// TwinCAT 3 PLC project Library
// Title: lcls-twincat-motion-abstraction
// Company: SLAC
// Author: YS Mandza
// ProjectVersion: 1.0.0
// Description: Motion Abstraction
// ProgramVersion: 3.1.4026.17
// libraries:
//   LCLS General, * (SLAC)
//   Tc2_EtherCAT, * (Beckhoff Automation GmbH)
//   Tc2_MC2, * (Beckhoff Automation GmbH)
//   Tc2_Standard, * (Beckhoff Automation GmbH)
//   Tc2_System, * (Beckhoff Automation GmbH)
//   Tc2_Utilities, * (Beckhoff Automation GmbH)
//   TcUnit, * (www.tcunit.org)
// project tree:
//   / DemoTask.TcTTO, PlcTask.TcTTO, UnitTestTask.TcTTO (not stored)
//   DUTs/ E_LCLSMotionError.TcDUT (not stored), E_MotionLogLevel.TcDUT, MOTION_LOGGER_MSG.TcDUT, ST_ExtendedMotionStatus.TcDUT, E_HomeStates.TcDUT (not stored), E_Module.TcDUT (not stored), ST_MotionStatus.TcDUT (not stored), ENUM_StageEnableMode.TcDUT (not stored), E_DS402HomingMethod.TcDUT (not stored), E_DS402OpMode.TcDUT (not stored), E_EpicsHomeCmd.TcDUT, E_EpicsMotorCmd.TcDUT, E_MoveMode.TcDUT (not stored), E_MoveState.TcDUT, E_StageBrakeMode.TcDUT, E_StageEnableMode.TcDUT (not stored), ST_AxisParameterSetExposed.TcDUT (not stored), ST_DS402Drive.TcDUT, ST_DS402DriveStatus.TcDUT (not stored), ST_AxisStatus.TcDUT (not stored), ST_MotionCommand.TcDUT (not stored), ST_MotionLogMessage.TcDUT, ST_MoveRequestStatus.TcDUT (not stored)
//   POUs/FBs/Common/ FB_EncoderScaling.TcPOU (not stored), FB_EpicsMotionParamsStatus.TcPOU (not stored), FB_EpicsMoveRequest.TcPOU, FB_LimSwStatus.TcPOU (not stored), FB_MotionDrive.TcPOU, FB_MotionDriveStateMachine.TcPOU (not stored), FB_MotionInterlocksCommon.TcPOU (not stored), FB_MotionInterlocksLimSw.TcPOU (not stored), FB_MotionLogger.TcPOU, FB_PersistentDataStorage.TcPOU (not stored)
//   POUs/FBs/Containers/ FB_MotionStageNC.TcPOU
//   POUs/FBs/DS402/ FB_HomeDS402.TcPOU (not stored) (excluded from build)
//   POUs/FBs/NC/ FB_AxisStatusNC.TcPOU (not stored) (excluded from build), FB_BacklashCompensationNC.TcPOU (not stored), FB_BrakeNC.TcPOU (not stored), FB_HaltNC.TcPOU (not stored), FB_HomeNC.TcPOU (not stored), FB_MotionAxisNC.TcPOU (not stored), FB_MoveAbsoluteNC.TcPOU (not stored), FB_ParamsSaveRestoreNC.TcPOU, FB_PowerInterlockNC.TcPOU (not stored), FB_PowerNC.TcPOU (not stored), FB_ReadParameterNC.TcPOU (not stored), FB_ResetNC.TcPOU (not stored), FB_WriteParameterNC.TcPOU (not stored)
//   POUs/ITFs/ I_AxisStatus.TcIO (not stored), I_BacklashCompensation.TcIO (not stored), I_Brake.TcIO (not stored), I_DS402GenericDrive.TcIO (not stored), I_EncoderScaling.TcIO (not stored), I_EpicsMotionParamsStatus.TcIO (not stored), I_Error.TcIO (not stored), I_Halt.TcIO, I_Home.TcIO (not stored), I_HomeDS402.TcIO (not stored), I_LimSwStatus.TcIO (not stored), I_MotionAxis.TcIO (not stored), I_MotionAxisDS402.TcIO (not stored), I_MotionDrive.TcIO (not stored), I_MotionInterlocks.TcIO (not stored), I_MotionInterlocksCommon.TcIO (not stored), I_MotionLogger.TcIO, I_MotionStage.TcIO (not stored), I_MoveAbsolute.TcIO (not stored), I_MoveRequest.TcIO, I_ParamsSaveRestore.TcIO, I_PersistentDataStorage.TcIO (not stored), I_Power.TcIO (not stored), I_ReadParameter.TcIO (not stored), I_Reset.TcIO (not stored), I_StateMachine.TcIO (not stored), I_Status.TcIO (not stored), I_StatusEx.TcIO (not stored), I_WriteParameter.TcIO (not stored)
//   Test/Containers/ FB_MotionStageNC_Test.TcPOU
//   Test/Interlok/ FB_MotionInterlocksCommon_Test.TcPOU, FB_MotionInterlocksLimSw_Test.TcPOU
//   Test/ HARD_TEST.TcPOU (not stored), PRG_TEST.TcPOU (not stored), CONTAINER_TEST.TcPOU (not stored)
//   Test/Orchetration/ FB_BrakeNC_Test.TcPOU (not stored), FB_MotionDriveStateMachine_Test.TcPOU, FB_MotionDrive_Test.TcPOU (not stored), FB_MoveRequest_Test.TcPOU
//   Test/NC/ FB_NcMotionBlocks_Test.TcPOU, FB_MotionAxisNC_Test.TcPOU
//   Test/TestDouble/ FB_AxisStatusNC_TestDouble.TcPOU (not stored), FB_BacklashCompensationNC_TestDouble.TcPOU (not stored), FB_Brake_TestDouble.TcPOU (not stored), FB_EncoderScalingNC_TestDouble.TcPOU (not stored), FB_EpicsMotionParamsStatus_TestDouble.TcPOU (not stored), FB_HaltNC_TestDouble.TcPOU, FB_HomeNC_TestDouble.TcPOU (not stored), FB_LimSwStatus_testDouble.TcPOU (not stored), FB_MotionAxisDS402_TestDouble.TcPOU, FB_MotionAxisNC_TestDouble.TcPOU (not stored), FB_StateMachine_TestDouble.TcPOU (not stored), FB_MotionInterlocksCommon_TestDouble.TcPOU (not stored), FB_MotionInterlocksLimSw_TestDouble.TcPOU, FB_MotionLogger_TestDouble.TcPOU, FB_MoveAbsoluteNC_TestDouble.TcPOU, FB_MoveRequest_TestDouble.TcPOU (not stored), FB_ParamSaveRestoreNC_TestDouble.TcPOU, FB_PersistentDataStorage_TestDouble.TcPOU, FB_PowerNC_TestDouble.TcPOU (not stored), FB_ReadParameterNC_TestDouble.TcPOU (not stored), FB_ResetNC_TestDouble.TcPOU, FB_WriteParameterNC_TestDouble.TcPOU (not stored)
//   Test/Utils/ FB_MotionLogger_Test.TcPOU (not stored)
//   VISUs/ motion.TcCD (not stored)
// real-time tasks:
//   TASK PlcTask: cycle T#10ms, priority 1, ADS port 350
//   TASK UnitTestTask: cycle T#10ms, priority 20, ADS port 351
//   TASK Demo: cycle T#10ms, priority 2, ADS port 352
// motion (NC):
//   TASK NC-Task 1 SAF: cycle T#2ms, priority 4, ADS port 501
//   TASK NC-Task 1 SVB: cycle T#10ms, priority 8, ADS port 511
//   AXIS Axis_HomeNC_Test8 (id 15)
//     OtherSettings: AllowMotionCmdToSlave=true
//     encoder EncType=1
//     drive DrvType=5
//       Analog: TorqueSetpointScale=10, ScaleFactorActTorque=0.1
//       TimeComp: TaskDelayCycles=1
//     controller CtrType=1
//       CtrPara: PriorControlFactor=1
//         Observer: BandWidth=20
//   AXIS Axis_HomeNC_Test7 (id 14)
//     OtherSettings: AllowMotionCmdToSlave=true
//     encoder EncType=1
//     drive DrvType=5
//       Analog: TorqueSetpointScale=10, ScaleFactorActTorque=0.1
//       TimeComp: TaskDelayCycles=1
//     controller CtrType=1
//       CtrPara: PriorControlFactor=1
//         Observer: BandWidth=20
//   AXIS Axis_HomeNC_Test6 (id 2)
//     OtherSettings: AllowMotionCmdToSlave=true
//     encoder EncType=1
//     drive DrvType=5
//       Analog: TorqueSetpointScale=10, ScaleFactorActTorque=0.1
//       TimeComp: TaskDelayCycles=1
//     controller CtrType=1
//       CtrPara: PriorControlFactor=1
//         Observer: BandWidth=20
//   AXIS Axis_HomeNC_Test5 (id 7)
//     OtherSettings: AllowMotionCmdToSlave=true
//     encoder EncType=1
//     drive DrvType=5
//       Analog: TorqueSetpointScale=10, ScaleFactorActTorque=0.1
//       TimeComp: TaskDelayCycles=1
//     controller CtrType=1
//       CtrPara: PriorControlFactor=1
//         Observer: BandWidth=20
//   AXIS Axis_HomeNC_Test4 (id 6)
//     OtherSettings: AllowMotionCmdToSlave=true
//     encoder EncType=1
//     drive DrvType=5
//       Analog: TorqueSetpointScale=10, ScaleFactorActTorque=0.1
//       TimeComp: TaskDelayCycles=1
//     controller CtrType=1
//       CtrPara: PriorControlFactor=1
//         Observer: BandWidth=20
//   AXIS Axis_HomeNC_Test3 (id 5)
//     OtherSettings: AllowMotionCmdToSlave=true
//     encoder EncType=1
//     drive DrvType=5
//       Analog: TorqueSetpointScale=10, ScaleFactorActTorque=0.1
//       TimeComp: TaskDelayCycles=1
//     controller CtrType=1
//       CtrPara: PriorControlFactor=1
//         Observer: BandWidth=20
//   AXIS Axis_HomeNC_Test2 (id 4)
//     Velo: RefSearch=500, RefSync=500
//     OtherSettings: AllowMotionCmdToSlave=true
//     encoder EncType=1
//     drive DrvType=5
//       Analog: TorqueSetpointScale=10, ScaleFactorActTorque=0.1
//       TimeComp: TaskDelayCycles=1
//     controller CtrType=1
//       CtrPara: PriorControlFactor=1
//         Observer: BandWidth=20
//   AXIS Axis_HomeNC_Test1 (id 3)
//     OtherSettings: AllowMotionCmdToSlave=true
//     encoder EncType=1
//     drive DrvType=5
//       Analog: TorqueSetpointScale=10, ScaleFactorActTorque=0.1
//       TimeComp: TaskDelayCycles=1
//     controller CtrType=1
//       CtrPara: PriorControlFactor=1
//         Observer: BandWidth=20
//   AXIS Axis_McMotionBlocks_Test1 (id 9)
//     OtherSettings: AllowMotionCmdToSlave=true
//     encoder EncType=1
//     drive DrvType=5
//       Analog: TorqueSetpointScale=10, ScaleFactorActTorque=0.1
//       TimeComp: TaskDelayCycles=1
//     controller CtrType=1
//       CtrPara: PriorControlFactor=1
//         Observer: BandWidth=20
//   AXIS Axis_McMotionBlocks_Test2 (id 10)
//     OtherSettings: AllowMotionCmdToSlave=true
//     encoder EncType=1
//     drive DrvType=5
//       Analog: TorqueSetpointScale=10, ScaleFactorActTorque=0.1
//       TimeComp: TaskDelayCycles=1
//     controller CtrType=1
//       CtrPara: PriorControlFactor=1
//         Observer: BandWidth=20
//   AXIS Axis_McMotionBlocks_Test3 (id 11)
//     OtherSettings: AllowMotionCmdToSlave=true
//     encoder EncType=1
//     drive DrvType=5
//       Analog: TorqueSetpointScale=10, ScaleFactorActTorque=0.1
//       TimeComp: TaskDelayCycles=1
//     controller CtrType=1
//       CtrPara: PriorControlFactor=1
//         Observer: BandWidth=20
//   AXIS Axis_McMotionBlocks_Test4 (id 12)
//     OtherSettings: AllowMotionCmdToSlave=true
//     encoder EncType=1
//     drive DrvType=5
//       Analog: TorqueSetpointScale=10, ScaleFactorActTorque=0.1
//       TimeComp: TaskDelayCycles=1
//     controller CtrType=1
//       CtrPara: PriorControlFactor=1
//         Observer: BandWidth=20
//   AXIS Axis_McMotionBlocks_Test8 (id 17)
//     OtherSettings: AllowMotionCmdToSlave=true
//     encoder EncType=1
//       ActPosCorrection: Enable=true
//     drive DrvType=5
//       Analog: TorqueSetpointScale=10, ScaleFactorActTorque=0.1
//       TimeComp: TaskDelayCycles=1
//     controller CtrType=1
//       CtrPara: PriorControlFactor=1
//         Observer: BandWidth=20
//   AXIS Axis_McMotionBlocks_Test7 (id 1)
//     OtherSettings: AllowMotionCmdToSlave=true
//     encoder EncType=1
//       ActPosCorrection: Enable=true
//     drive DrvType=5
//       Analog: TorqueSetpointScale=10, ScaleFactorActTorque=0.1
//       TimeComp: TaskDelayCycles=1
//     controller CtrType=1
//       CtrPara: PriorControlFactor=1
//         Observer: BandWidth=20
//   AXIS Axis_McMotionBlocks_Test6 (id 16)
//     OtherSettings: AllowMotionCmdToSlave=true
//     encoder EncType=1
//       ActPosCorrection: Enable=true
//     drive DrvType=5
//       Analog: TorqueSetpointScale=10, ScaleFactorActTorque=0.1
//       TimeComp: TaskDelayCycles=1
//     controller CtrType=1
//       CtrPara: PriorControlFactor=1
//         Observer: BandWidth=20
//   AXIS Axis_McMotionBlocks_Test5 (id 13)
//     OtherSettings: AllowMotionCmdToSlave=true
//     encoder EncType=1
//     drive DrvType=5
//       Analog: TorqueSetpointScale=10, ScaleFactorActTorque=0.1
//       TimeComp: TaskDelayCycles=1
//     controller CtrType=1
//       CtrPara: PriorControlFactor=1
//         Observer: BandWidth=20
//   AXIS Axis_Hard_Test (id 8)
//     Velo: RefSync=100
//     OtherSettings: AllowMotionCmdToSlave=true
//     encoder EncType=1
//       ActPosCorrection: Enable=true
//     drive DrvType=5
//       Analog: TorqueSetpointScale=10, ScaleFactorActTorque=0.1
//       TimeComp: TaskDelayCycles=1
//     controller CtrType=1
//       CtrPara: PriorControlFactor=1
//         Observer: BandWidth=20
// variable links:
//   motion/motion Instance <-> NC-Task 1 SAF/Axes/Axis_Hard_Test
//     DemoTask Inputs/NcAxis_GVL.NC.NcToPlc <-> Outputs/ToPlc
//     DemoTask Outputs/NcAxis_GVL.NC.PlcToNc <-> Inputs/FromPlc
//   motion/motion Instance <-> NC-Task 1 SAF/Axes/Axis_HomeNC_Test1
//     UnitTestTask Inputs/PRG_TEST.fb_HomeNC_Test.fbAxisRef[1].NcToPlc <-> Outputs/ToPlc
//     UnitTestTask Outputs/PRG_TEST.fb_HomeNC_Test.fbAxisRef[1].PlcToNc <-> Inputs/FromPlc
//   motion/motion Instance <-> NC-Task 1 SAF/Axes/Axis_HomeNC_Test2
//     UnitTestTask Inputs/PRG_TEST.fb_HomeNC_Test.fbAxisRef[2].NcToPlc <-> Outputs/ToPlc
//     UnitTestTask Outputs/PRG_TEST.fb_HomeNC_Test.fbAxisRef[2].PlcToNc <-> Inputs/FromPlc
//   motion/motion Instance <-> NC-Task 1 SAF/Axes/Axis_HomeNC_Test3
//     UnitTestTask Inputs/PRG_TEST.fb_HomeNC_Test.fbAxisRef[3].NcToPlc <-> Outputs/ToPlc
//     UnitTestTask Outputs/PRG_TEST.fb_HomeNC_Test.fbAxisRef[3].PlcToNc <-> Inputs/FromPlc
//   motion/motion Instance <-> NC-Task 1 SAF/Axes/Axis_HomeNC_Test4
//     UnitTestTask Inputs/PRG_TEST.fb_HomeNC_Test.fbAxisRef[4].NcToPlc <-> Outputs/ToPlc
//     UnitTestTask Outputs/PRG_TEST.fb_HomeNC_Test.fbAxisRef[4].PlcToNc <-> Inputs/FromPlc
//   motion/motion Instance <-> NC-Task 1 SAF/Axes/Axis_HomeNC_Test5
//     UnitTestTask Inputs/PRG_TEST.fb_HomeNC_Test.fbAxisRef[5].NcToPlc <-> Outputs/ToPlc
//     UnitTestTask Outputs/PRG_TEST.fb_HomeNC_Test.fbAxisRef[5].PlcToNc <-> Inputs/FromPlc
//   motion/motion Instance <-> NC-Task 1 SAF/Axes/Axis_HomeNC_Test6
//     UnitTestTask Inputs/PRG_TEST.fb_HomeNC_Test.fbAxisRef[6].NcToPlc <-> Outputs/ToPlc
//     UnitTestTask Outputs/PRG_TEST.fb_HomeNC_Test.fbAxisRef[6].PlcToNc <-> Inputs/FromPlc
//   motion/motion Instance <-> NC-Task 1 SAF/Axes/Axis_HomeNC_Test7
//     UnitTestTask Inputs/PRG_TEST.fb_HomeNC_Test.fbAxisRef[7].NcToPlc <-> Outputs/ToPlc
//     UnitTestTask Outputs/PRG_TEST.fb_HomeNC_Test.fbAxisRef[7].PlcToNc <-> Inputs/FromPlc
//   motion/motion Instance <-> NC-Task 1 SAF/Axes/Axis_HomeNC_Test8
//     UnitTestTask Inputs/PRG_TEST.fb_HomeNC_Test.fbAxisRef[8].NcToPlc <-> Outputs/ToPlc
//     UnitTestTask Outputs/PRG_TEST.fb_HomeNC_Test.fbAxisRef[8].PlcToNc <-> Inputs/FromPlc
//   motion/motion Instance <-> NC-Task 1 SAF/Axes/Axis_McMotionBlocks_Test1
//     UnitTestTask Inputs/PRG_TEST.fb_McMotionBlocks_Test.fbAxisRef[1].NcToPlc <-> Outputs/ToPlc
//     UnitTestTask Outputs/PRG_TEST.fb_McMotionBlocks_Test.fbAxisRef[1].PlcToNc <-> Inputs/FromPlc
//   motion/motion Instance <-> NC-Task 1 SAF/Axes/Axis_McMotionBlocks_Test2
//     UnitTestTask Inputs/PRG_TEST.fb_McMotionBlocks_Test.fbAxisRef[2].NcToPlc <-> Outputs/ToPlc
//     UnitTestTask Outputs/PRG_TEST.fb_McMotionBlocks_Test.fbAxisRef[2].PlcToNc <-> Inputs/FromPlc
//   motion/motion Instance <-> NC-Task 1 SAF/Axes/Axis_McMotionBlocks_Test3
//     UnitTestTask Inputs/PRG_TEST.fb_McMotionBlocks_Test.fbAxisRef[3].NcToPlc <-> Outputs/ToPlc
//     UnitTestTask Outputs/PRG_TEST.fb_McMotionBlocks_Test.fbAxisRef[3].PlcToNc <-> Inputs/FromPlc
//   motion/motion Instance <-> NC-Task 1 SAF/Axes/Axis_McMotionBlocks_Test4
//     UnitTestTask Inputs/PRG_TEST.fb_McMotionBlocks_Test.fbAxisRef[4].NcToPlc <-> Outputs/ToPlc
//     UnitTestTask Outputs/PRG_TEST.fb_McMotionBlocks_Test.fbAxisRef[4].PlcToNc <-> Inputs/FromPlc
//   motion/motion Instance <-> NC-Task 1 SAF/Axes/Axis_McMotionBlocks_Test5
//     UnitTestTask Inputs/PRG_TEST.fb_McMotionBlocks_Test.fbAxisRef[5].NcToPlc <-> Outputs/ToPlc
//     UnitTestTask Outputs/PRG_TEST.fb_McMotionBlocks_Test.fbAxisRef[5].PlcToNc <-> Inputs/FromPlc
//   motion/motion Instance <-> NC-Task 1 SAF/Axes/Axis_McMotionBlocks_Test6
//     UnitTestTask Inputs/PRG_TEST.fb_McMotionBlocks_Test.fbAxisRef[6].NcToPlc <-> Outputs/ToPlc
//     UnitTestTask Outputs/PRG_TEST.fb_McMotionBlocks_Test.fbAxisRef[6].PlcToNc <-> Inputs/FromPlc
//   motion/motion Instance <-> NC-Task 1 SAF/Axes/Axis_McMotionBlocks_Test7
//     UnitTestTask Inputs/PRG_TEST.fb_McMotionBlocks_Test.fbAxisRef[7].NcToPlc <-> Outputs/ToPlc
//     UnitTestTask Outputs/PRG_TEST.fb_McMotionBlocks_Test.fbAxisRef[7].PlcToNc <-> Inputs/FromPlc
//   motion/motion Instance <-> NC-Task 1 SAF/Axes/Axis_McMotionBlocks_Test8
//     UnitTestTask Inputs/PRG_TEST.fb_McMotionBlocks_Test.fbAxisRef[8].NcToPlc <-> Outputs/ToPlc
//     UnitTestTask Outputs/PRG_TEST.fb_McMotionBlocks_Test.fbAxisRef[8].PlcToNc <-> Inputs/FromPlc

CONFIGURATION Library
    RESOURCE PLC ON TwinCAT3
        TASK DemoTask(INTERVAL := T#10ms, PRIORITY := 2);
        TASK PlcTask(INTERVAL := T#10ms, PRIORITY := 1);
        PROGRAM CONTAINER_TEST WITH DemoTask : CONTAINER_TEST;
        PROGRAM HARD_TEST WITH PlcTask : HARD_TEST;
    END_RESOURCE
END_CONFIGURATION

// ---- DUTs/E_MotionLogLevel.TcDUT
{attribute 'qualified_only'}
{attribute 'strict'}
{attribute 'to_string'}
TYPE E_MotionLogLevel :
(
	WARNING := 0,
	ERROR := 1,
	INFO := 2
);
END_TYPE

// ---- DUTs/MOTION_LOGGER_MSG.TcDUT
TYPE MOTION_LOGGER_MSG : STRING(128); END_TYPE

// ---- DUTs/ST_ExtendedMotionStatus.TcDUT
TYPE ST_ExtendedMotionStatus :
STRUCT
	bMotionAxisError : BOOL;
	nMotionAxisErrorId : UDINT;
	bInterlocksError : BOOL;
	nInterlocksError : UDINT;
	eDriveState : E_MoveState;
	bDriveWatchDogStatus : BOOL;
	bAbortDone : BOOL;
	bAborted : BOOL;
	bLimHomeDone : BOOL;
	bNewMoveReq : BOOL;
	bExecute : BOOL;
	bEnable : BOOL;
	bIdling : BOOL;
END_STRUCT
END_TYPE

// ---- DUTs/E_EpicsHomeCmd.TcDUT
{attribute 'qualified_only'}
{attribute 'strict'}
TYPE E_EpicsHomeCmd :
    // Defines the valid options for homing in FB_MotionStage
(
    LOW_LIMIT := 1, // Low limit switch
    HIGH_LIMIT := 2, // High limit switch
    HOME_VIA_LOW := 3, // Home switch via low switch
    HOME_VIA_HIGH := 4, // Home switch via high switch
    ABSOLUTE_SET := 15, // Set here to be fHomePosition
    // MCS2
    AUTOZERO := -1,
    CURRENT_POSITION_METHOD := 37,
    NONE := -99 // Do not home, ever
) INT := NONE;
END_TYPE

// ---- DUTs/E_EpicsMotorCmd.TcDUT
{attribute 'qualified_only'}
{attribute 'strict'}
TYPE E_EpicsMotorCmd :
    // Defines valid EPICS commands for nCommand
(
    JOG := 0,
    MOVE_VELOCITY := 1,
    MOVE_RELATIVE := 2,
    MOVE_ABSOLUTE := 3,
    MOVE_MODULO := 4,
    HOME := 10,
    GEAR := 30
)INT;
END_TYPE

// ---- DUTs/E_MoveState.TcDUT
{attribute 'qualified_only'}
{attribute 'to_string'}
TYPE E_MoveState :
(
    IDLING:=0,
    INIT:=10,
    STARTED:=20,
    IN_PROGRESS :=30,
    REACHED:=40,
    INTERRUPTED:=50,
    DONE:=60,
    ERROR:=-99
) INT;
END_TYPE

// ---- DUTs/E_StageBrakeMode.TcDUT
{attribute 'qualified_only'}
{attribute 'strict'}
TYPE E_StageBrakeMode :
    // Defines when to send the brake disengage signal in FB_MotionStage
(
    IF_ENABLED := 0, // Disengage brake when the motor is enabled
    IF_MOVING, // Disengage brake when the motor is moving
    NO_BRAKE // Do not change the brake state in FB_MotionStage
)INT;
END_TYPE

// ---- DUTs/ST_DS402Drive.TcDUT
TYPE ST_DS402Drive:
STRUCT
    (* Global variables for the TPDO data from the drive. Each one is linked to the respective TPDO channel. *)
    stDriveStatus 			AT %I*	: 	ST_DS402DriveStatus;
    nModeOfOperationDisplay AT %I*	: 	SINT;
    //nActualPosition 		AT %I*	: 	DINT;
    (*CSP drive mode*)
    nFollowingError 		AT %I*	: 	DINT;
    (* Global variables for the RPDO data to the drive. Each one is linked to the respective RPDO channel. *)
    //nDS402DriveControl		AT %Q*	:	UINT;
    // Connected to NC task Ctrl 1 and Ctrl 2
       nDS402DriveControlNC	AT %I*	:	UINT;
    // connected to I/O Task 'Control Word'
       nDS402DriveControl		AT %Q*	:	UINT;
    //nTargetPositionTmp 		AT %I* 	: 	DINT;
    nTargetPosition 		AT %Q* 	: 	DINT;
    nModeOfOperationNC 	AT %I* 	: 	SINT;
    nModeOfOperation 		AT %Q* 	: 	SINT;
    (* Global variables for the RPDO data to the drive. Each one is linked to the respective RPDO channel. *)
    nProfilVelocity 		AT %Q* 	: 	DINT;
    nProfilAcceleration		AT %Q* 	: 	DINT;
    nProfilDecceleration	AT %Q* 	: 	DINT;
    nVelocityActualValue	AT %Q* 	: 	DINT;
    (* Global variables for the TPDO data from the drive. Each one is linked to the respective TPDO channel. *)
    nScantargetPosition		AT %Q*	: 	DINT;
    uScantargetVelocity		AT %Q*	: 	ULINT;

    {attribute 'pytmc' := '
        pv: PLC:nChanStep
        io: io
        field: DESC SmartAct: Open Loop Step Count
    '}
    nChanStep			: DINT;

    {attribute 'pytmc' := '
        pv: PLC:nChanStepFreq
        io: io
        field: DESC SmartAct: Open Loop Step Freq
    '}
    nChanStepFreq		: UINT;

    {attribute 'pytmc' := '
        pv: PLC:nChanStepAmp
        io: io
        field: DESC SmartAct: Open Loop Step Amp
    '}
    nChanStepAmp		: UINT;

    // timeout for holding actual position in close loop mode
    {attribute 'pytmc' := '
        pv: PLC:nHoldTime
        io: io
        field: DESC SmartAct: Set servo mode hold time
    '}
    nHoldTime						: UDINT := 10000;

    {attribute 'pytmc' := '
        pv: PLC:bServo
        io: io
        field: ZNAM DISABLE
        field: ONAM ENABLE
        field: DESC Used to disable close loop mode
    '}
    bServo							: BOOL := TRUE;

    (* NetId of EtherCAT Master *)
    arNetId  				AT %I*	: 	AMSNETID;
    (* Port Number of EtherCAT Slave *)
    nSlaveAddr 				AT %I* 	: 	UINT;

END_STRUCT
END_TYPE

// ---- DUTs/ST_MotionLogMessage.TcDUT
TYPE ST_MotionLogMessage :
STRUCT
    sSource : STRING(64);
    sMessage : MOTION_LOGGER_MSG;
    sTimestamp : STRING(16);
    eLevel : E_MotionLogLevel;
END_STRUCT
END_TYPE

// ---- POUs/ITFs/I_Halt.TcIO
INTERFACE I_Halt EXTENDS I_StatusEx

METHOD ClearStatus
VAR_INPUT
END_VAR
END_METHOD

PROPERTY CommandHalt : BOOL
SET
END_SET
END_PROPERTY

METHOD Halt
VAR_INPUT
    Deceleration : LREAL := 0.0;
    Jerk : LREAL := 0.0;
    BufferMode	: MC_BufferMode := MC_BufferMode.MC_Aborting;
END_VAR
END_METHOD

END_INTERFACE

// ---- POUs/ITFs/I_MotionLogger.TcIO
INTERFACE I_MotionLogger

METHOD Clear
VAR_INPUT
END_VAR
END_METHOD

METHOD ErrorCodeLookup : STRING
VAR_INPUT
	 nErrorId: UDINT;
END_VAR
END_METHOD

METHOD GetAllMessages : STRING(1024)
END_METHOD

METHOD GetMessageCount : UINT
VAR_OUTPUT
    nCount : UINT;
END_VAR
END_METHOD

METHOD Logger
VAR_INPUT
    Message : STRING;
    Level   : E_MotionLogLevel := E_MotionLogLevel.INFO;
    Source  : STRING := '';
END_VAR
END_METHOD

PROPERTY Name : STRING
GET
END_GET
END_PROPERTY

END_INTERFACE

// ---- POUs/ITFs/I_MoveRequest.TcIO
INTERFACE I_MoveRequest

METHOD ClearMoveRequest
END_METHOD

METHOD ClearMoveRequestErrors
VAR_INPUT
END_VAR
END_METHOD

PROPERTY EnableMode : ENUM_StageEnableMode
GET
END_GET
SET
END_SET
END_PROPERTY

METHOD InitMoveRequest
VAR_INPUT
END_VAR
END_METHOD

METHOD IsValidHomeCmd : BOOL
VAR_INPUT
    CmdData : INT;
END_VAR
END_METHOD

METHOD MoveRequest
VAR_INPUT
	// From Axis through the drive
	EnableDone	: BOOL;
	// From Interlock through the drive
	MoveOk  : BOOL;
END_VAR
END_METHOD

METHOD MoveRequestCompleted
VAR_INPUT
	MoveDone : BOOL;
	HomeDone : BOOL;
END_VAR
END_METHOD

METHOD MoveRequestDone
VAR_INPUT
	Done : BOOL;
END_VAR
END_METHOD

METHOD MoveRequestError
VAR_INPUT
Error :BOOL;
ErrorId :UDINT;
ErrorMessage:T_MAXSTRING;
END_VAR
END_METHOD

METHOD ResetMoveEnable : BOOL
END_METHOD

METHOD RestoreSettings
VAR_INPUT
	RestoreDone : BOOL;
	SavedPosition : LREAL;
END_VAR
END_METHOD

PROPERTY Status : REFERENCE TO ST_MoveRequestStatus
GET
END_GET
END_PROPERTY

METHOD StopMoveRequest
VAR_INPUT
END_VAR
END_METHOD

END_INTERFACE

// ---- POUs/ITFs/I_ParamsSaveRestore.TcIO
INTERFACE I_ParamsSaveRestore EXTENDS I_Status

METHOD RestoreAxisParams
VAR_INPUT
END_VAR
END_METHOD

METHOD SaveAxisParams
VAR_INPUT
    Enable : BOOL;
END_VAR
END_METHOD

PROPERTY SavedPosition : LREAL
GET
END_GET
END_PROPERTY

END_INTERFACE

// ---- POUs/FBs/Common/FB_EpicsMoveRequest.TcPOU
(*Implements MoveRequest interface for EPICS Motor*)
FUNCTION_BLOCK FB_EpicsMoveRequest IMPLEMENTS I_MoveRequest
VAR
   // EPICS Interface
    {attribute 'no_copy'}
    stMotionCommand : REFERENCE TO ST_MotionCommand;
	{attribute 'no_copy'}
	stMotionStatus:  REFERENCE TO ST_MotionStatus;
	
    eEnableMode: E_StageEnableMode:=E_StageEnableMode.DURING_MOTION;
    {attribute 'hide'}
    eHomeMode	: E_EpicsHomeCmd := E_EpicsHomeCmd.NONE;
    {attribute 'hide'}
    bEnableDone : BOOL;
    {attribute 'hide'}
    bMoveOk: BOOL;
    (* non epics*)
    {attribute 'hide'}
    bExecute : BOOL;
    {attribute 'hide'}
    rtMoveCmdShortcut: R_TRIG;
    {attribute 'hide'}
    rtHomeCmdShortcut: R_TRIG;
    {attribute 'hide'}
    rtEnableMode: R_TRIG;
    {attribute 'hide'}
    rtNewMoveReq: R_TRIG;
    {attribute 'hide'}
    rtUserExec: R_TRIG;
    {attribute 'hide'}
    rtExec : R_TRIG;
    {attribute 'hide'}
    stMotionRequestStatus : ST_MoveRequestStatus;
    {attribute 'hide'}
    ftStopExec: F_TRIG;
    {attribute 'hide'}
    eRestoreSettingsState : ( RestoreSettingWaiting:=0, RestoreSettingDone:=1);
	rtExecute : R_TRIG;
END_VAR

// --- Validate command and status references ---
IF NOT __ISVALIDREF(stMotionCommand) OR NOT __ISVALIDREF(stMotionStatus) THEN
   RETURN;
END_IF

// --- Handle PLC shortcut commands (testing/circumvention logic) ---
rtMoveCmdShortcut(CLK := stMotionCommand.bMoveCmd);
rtHomeCmdShortcut(CLK := stMotionCommand.bHomeCmd);

// --- Rising edge of move command: issue MOVE_ABSOLUTE ---
IF rtMoveCmdShortcut.Q AND NOT bExecute THEN
    bExecute := TRUE;
    stMotionCommand.nCommand := E_EpicsMotorCmd.MOVE_ABSOLUTE;

// --- Rising edge of home command: validate and set HOME mode ---
ELSIF rtHomeCmdShortcut.Q AND NOT bExecute THEN
    IF IsValidHomeCmd(stMotionCommand.nCmdData) THEN
        IF stMotionCommand.nCmdData = E_EpicsHomeCmd.NONE THEN
            bExecute := FALSE; // Do not execute
        ELSE
            bExecute := TRUE;  // Valid home: enable
        END_IF
        stMotionCommand.nCommand := E_EpicsMotorCmd.HOME;
    END_IF
END_IF

// --- User/EPICS main exec entry ---
rtUserExec(CLK := bExecute);

// --- New move request: rising edge, axis not busy, no error, and interlocks OK ---
stMotionRequestStatus.bNewMoveReq S= NOT stMotionStatus.bBusy AND rtUserExec.Q AND NOT stMotionStatus.bError AND bMoveOk;

// --- New move stays active until execute ends or error occurs ---
stMotionRequestStatus.bNewMoveReq R= NOT bExecute OR stMotionStatus.bError;

// --- Prepare disable on end of move ---
stMotionRequestStatus.bPrepareDisable R= stMotionRequestStatus.bNewMoveReq;
rtNewMoveReq(CLK := stMotionRequestStatus.bNewMoveReq);

// --- Latch command data/type at queue entry, and check homing prerequisites ---
IF rtUserExec.Q THEN
    stMotionRequestStatus.nCmdData := stMotionCommand.nCmdData;
    stMotionRequestStatus.nCommand := stMotionCommand.nCommand;
    IF NOT stMotionCommand.bHomeCmd THEN
        IF eHomeMode <> E_EpicsHomeCmd.NONE AND NOT stMotionStatus.bHomed THEN
            stMotionStatus.sErrorMessage := 'Axis homing mode set, but homing routine pending';
        END_IF
    END_IF
END_IF

// --- Enable logic based on requested enable mode ---
rtEnableMode(CLK := (eEnableMode = E_StageEnableMode.DURING_MOTION));
CASE eEnableMode OF
    E_StageEnableMode.ALWAYS:
        stMotionRequestStatus.bEnable := NOT stMotionStatus.bError AND bMoveOk;
    E_StageEnableMode.DURING_MOTION:
        IF rtEnableMode.Q THEN
            stMotionRequestStatus.bEnable := FALSE; // DuringMotion disables enable on falling edge
        END_IF
        IF rtNewMoveReq.Q THEN
            stMotionRequestStatus.bEnable S= stMotionRequestStatus.bNewMoveReq;
        END_IF
END_CASE

// --- Execute if: not error, Execute set, and axis ready ---
stMotionRequestStatus.bExecute := NOT stMotionStatus.bError AND bExecute AND bEnableDone;
stMotionRequestStatus.bExecHome := stMotionRequestStatus.bExecute AND stMotionRequestStatus.nCommand = E_EpicsMotorCmd.HOME;
stMotionRequestStatus.bExecMove := stMotionRequestStatus.bExecute AND NOT stMotionRequestStatus.bExecHome;

// --- Latch axis busy at execute (clear done, busy, error) ---
rtExecute(CLK := bExecute);
IF rtExecute.Q THEN
    InitMoveRequest();
END_IF

// --- Clear local/EPICS interface --- 
stMotionCommand.bMoveCmd := FALSE;
stMotionCommand.bHomeCmd := FALSE;

// --- Prepare to disable at the end of execution (on falling edge) ---
ftStopExec(CLK := bExecute);
stMotionRequestStatus.bPrepareDisable S= (eEnableMode = E_StageEnableMode.DURING_MOTION) AND ftStopExec.Q;

// --- Reset error message on busy; optional: else show string on error condition ---
IF stMotionStatus.bBusy THEN
    stMotionStatus.sErrorMessage := '';
END_IF

METHOD PUBLIC CallAfterInit
VAR_INPUT
    stMotionCommand : REFERENCE TO ST_MotionCommand;
	stMotionStatus:  REFERENCE TO ST_MotionStatus;
END_VAR
THIS^.stMotionCommand REF=stMotionCommand;
THIS^.stMotionStatus REF=stMotionStatus;
END_METHOD

METHOD ClearMoveRequest
// falling edge here when target is reached, move halted
bExecute := FALSE;
stMotionStatus.bDone := FALSE;
stMotionStatus.bBusy := FALSE;
// release the cmds
stMotionCommand.bHomeCmd:=FALSE;
stMotionCommand.bMoveCmd:=FALSE;
END_METHOD

METHOD ClearMoveRequestErrors
stMotionStatus.bError := FALSE;
stMotionStatus.nErrorId := 0;
stMotionStatus.sErrorMessage := '';
stMotionRequestStatus.bExecute := FALSE;
END_METHOD

PROPERTY EnableMode : ENUM_StageEnableMode
GET
EnableMode := eEnableMode;
END_GET
SET
eEnableMode := EnableMode;
END_SET
END_PROPERTY

//FB_Init is always available implicitly and it is used primarily for initialization.
//The return value is not evaluated. For a specific influence, you can also declare the
//methods explicitly and provide additional code there with the standard initialization
//code. You can evaluate the return value.
METHOD FB_Init: BOOL
VAR_INPUT
    bInitRetains: BOOL; // TRUE: the retain variables are initialized (reset warm / reset cold)
    bInCopyCode: BOOL;  // TRUE: the instance will be copied to the copy code afterward (online change)
    stMotionCommand : REFERENCE TO ST_MotionCommand;
	stMotionStatus:  REFERENCE TO ST_MotionStatus;
END_VAR
THIS^.stMotionCommand REF=stMotionCommand;
THIS^.stMotionStatus REF=stMotionStatus;
END_METHOD

METHOD InitMoveRequest
stMotionStatus.bBusy := TRUE;
stMotionStatus.bDone := FALSE;
// reset error flag
stMotionStatus.sErrorMessage := '';
END_METHOD

METHOD IsValidHomeCmd : BOOL
VAR_INPUT
    CmdData : INT;
END_VAR
CASE CmdData OF
    E_EpicsHomeCmd.LOW_LIMIT,
    E_EpicsHomeCmd.HIGH_LIMIT,
    E_EpicsHomeCmd.HOME_VIA_LOW,
    E_EpicsHomeCmd.HOME_VIA_HIGH,
    E_EpicsHomeCmd.ABSOLUTE_SET,
    E_EpicsHomeCmd.AUTOZERO,
    E_EpicsHomeCmd.CURRENT_POSITION_METHOD,
    E_EpicsHomeCmd.NONE:
        IsValidHomeCmd := TRUE;
    ELSE
        IsValidHomeCmd := FALSE;
END_CASE
END_METHOD

METHOD MoveRequest
VAR_INPUT
    // From Axis through the drive
    EnableDone	: BOOL;
    // From Interlock through the drive
    MoveOk  : BOOL;
END_VAR
THIS^.bMoveOk := MoveOk;
THIS^.bEnableDone := EnableDone;
END_METHOD

(*Internal use only purpose*)
METHOD INTERNAL MoveRequestCmds
VAR_INPUT
    (* From Drive*)
    HomeCmd		: BOOL;
    MoveCmd		: BOOL;
	MoveOk 		: BOOL;
	EnableDone  : BOOL;
    HomeMode	: INT := E_EpicsHomeCmd.NONE;
    EnableMode	: E_StageEnableMode :=  E_StageEnableMode.DURING_MOTION;
END_VAR
THIS^.stMotionCommand.bHomeCmd := HomeCmd;
THIS^.stMotionCommand.nCmdData := HomeMode;
THIS^.stMotionCommand.bMoveCmd	:= MoveCmd;
THIS^.bMoveOk := MoveOk;
THIS^.bEnableDone := EnableDone;
THIS^.eEnableMode := EnableMode;
END_METHOD

METHOD MoveRequestCompleted
VAR_INPUT
    MoveDone : BOOL;
    HomeDone : BOOL;
END_VAR
stMotionStatus.bHomed := HomeDone;
ClearMoveRequest();
MoveRequestDone(Done:=MoveDone OR HomeDone);
END_METHOD

METHOD MoveRequestDone
VAR_INPUT
    Done : BOOL;
END_VAR
stMotionStatus.bDone := Done;
END_METHOD

METHOD MoveRequestError
VAR_INPUT
    Error :BOOL;
    ErrorId :UDINT;
    ErrorMessage:T_MAXSTRING;
END_VAR
stMotionStatus.bError := Error;
stMotionStatus.nErrorId := ErrorId;
stMotionStatus.sErrorMessage:= ErrorMessage;

IF Error THEN
	ClearMoveRequest();
END_IF
END_METHOD

METHOD ResetMoveEnable : BOOL
IF stMotionRequestStatus.bPrepareDisable THEN
    IF THIS^.eEnableMode=E_StageEnableMode.DURING_MOTION THEN
        THIS^.stMotionRequestStatus.bEnable := FALSE;
		ResetMoveEnable := TRUE;
	ELSE
		ResetMoveEnable := FALSE;
    END_IF
    THIS^.stMotionRequestStatus.bPrepareDisable := FALSE;
END_IF
END_METHOD

METHOD RestoreSettings
VAR_INPUT
    RestoreDone : BOOL;
    SavedPosition : LREAL;
END_VAR
// no needed in production since the actual position is already set on the axis
// and epics status will get that last position
// use this to restore anything thats not an axisref paramter.

CASE eRestoreSettingsState OF
    RestoreSettingWaiting:
        IF RestoreDone THEN
            THIS^.stMotionCommand.fPosition := SavedPosition;
            eRestoreSettingsState := RestoreSettingDone;
        END_IF
    RestoreSettingDone:;

END_CASE
END_METHOD

PROPERTY INTERNAL RestoreSettingsState : UINT
GET
//RestoreSettingsState := eRestoreSettingsState;
END_GET
END_PROPERTY

PROPERTY Status : REFERENCE TO ST_MoveRequestStatus
GET
Status REF= stMotionRequestStatus;
END_GET
END_PROPERTY

METHOD StopMoveRequest
THIS^.bExecute := FALSE;
END_METHOD

END_FUNCTION_BLOCK

// ---- POUs/FBs/Common/FB_MotionDrive.TcPOU
FUNCTION_BLOCK FB_MotionDrive IMPLEMENTS I_MotionDrive
VAR
    stMotionCommand   : REFERENCE TO ST_MotionCommand;
    stMotionStatus    : REFERENCE TO ST_MotionStatus;
    stExMotionStatus  : REFERENCE TO ST_ExtendedMotionStatus;

    iAxis             : I_MotionAxis;         // Underlying axis logic (stepper, servo, simulated, etc.)
    iInterlocks       : I_MotionInterlocks;   // Interlocks interface for safety/hardware limits
    iLogger           : I_MotionLogger;       // Logging interface
    iMoveRequest      : I_MoveRequest;        // Move/home/stop request interface
    iStateMachine     : I_StateMachine;       // State coordination logic interface
    iBrake            : I_Brake;              // Brake interface

    bSaveAxisParams   : BOOL := TRUE;        // If axis parameters should be saved
    fbTimer           : TON;                  // Timer for internal delayed actions, etc.
    
    // Internal signals/state as needed
    bError            : BOOL;
    rtRestoreDone     : R_TRIG;
    nErrorId          : UDINT;
    sErrorMessage     : STRING;
END_VAR

// Restore Position Handling and Axis Parameter Save
rtRestoreDone(CLK := THIS^.iAxis.Status.bRestoreDone AND bSaveAxisParams);
IF rtRestoreDone.Q THEN
    THIS^.stMotionCommand.fPosition := THIS^.iAxis.Status.fSavedPosition;
END_IF

// Update Interlocks & Move Request Enable based on axis status and interlocks
iInterlocks.AxisStatus(
    HomeBusy           := iAxis.Status.bHomeBusy,
    PositiveDirection  := iAxis.Status.bPositiveMotionIsEnabled,
    NegativeDirection  := iAxis.Status.bNegativeMotionIsEnabled
);

iMoveRequest.MoveRequest(
    EnableDone := iAxis.AxisEnabled(),
    MoveOk     := iInterlocks.MoveOk
);

// Handle Halt (user stop only, not interlock or reset)
IF stMotionCommand.bHalt THEN
    THIS^.iMoveRequest.StopMoveRequest();
    
    IF iAxis.Status.bHomeBusy THEN
        iAxis.HomeAbortRecovery();
    END_IF

    // Use enum for command codes instead of magic numbers
    IF NOT stMotionCommand.bReset AND iAxis.Status.bBusy AND (
        (iMoveRequest.Status.nCommand = E_EpicsMotorCmd.HOME) OR
        (iMoveRequest.Status.nCommand = E_EpicsMotorCmd.MOVE_ABSOLUTE)
    ) THEN
        iAxis.Halt(Deceleration := stMotionCommand.fDeceleration);        
    END_IF

    stMotionCommand.bHalt := FALSE;
END_IF

// Handle Reset (clears move requests, errors, state machines, axis reset)
IF stMotionCommand.bReset THEN
    iMoveRequest.ClearMoveRequest();
    iMoveRequest.ClearMoveRequestErrors();
    iInterlocks.Reset();
    iStateMachine.Reset();

    IF iAxis.Status.bHomeBusy THEN
        iAxis.HomeAbortRecovery();
    END_IF

    iAxis.Reset();
    stMotionCommand.bReset := FALSE;
END_IF

// Axis Power Control
iAxis.Power(
    Enable           := iInterlocks.PowerEnabled,
    Enable_Positive  := iMoveRequest.Status.bExecHome OR iInterlocks.MoveForwardEnabled,
    Enable_Negative  := iMoveRequest.Status.bExecHome OR iInterlocks.MoveBackwardEnabled,
    Override         := 100.0,
    BufferMode       := MC_Aborting
);

// Interlock Drive Commands
iInterlocks.DriveCommands(
    MoveEnable := iMoveRequest.Status.bEnable,
    NewMoveReq := iMoveRequest.Status.bNewMoveReq
);

// Axis Parameters Handling
iAxis.ReadAxisParams(
    Enable       := TRUE,
    RefreshDelay := T#1S
);

iAxis.SaveAxisParams(
    Enable := bSaveAxisParams
);

// Error and Warning Status Handling (Axis > Interlock Error > Interlock Warning > None)
IF iAxis.Status.bError THEN
    THIS^.bError       := iAxis.Status.bError;
    THIS^.nErrorId     := iAxis.Status.nErrorID;
    THIS^.sErrorMessage:= iAxis.Status.sMessage;
ELSIF iInterlocks.Error THEN
    THIS^.bError       := iInterlocks.Error;
    THIS^.nErrorId     := iInterlocks.ErrorID;
    THIS^.sErrorMessage:= iInterlocks.Message;
ELSIF iInterlocks.Warning THEN
    THIS^.bError       := FALSE;
    THIS^.nErrorId     := 0;
    THIS^.sErrorMessage:= iInterlocks.Message;
ELSE
    THIS^.bError       := FALSE;
    THIS^.nErrorId     := 0;
    THIS^.sErrorMessage:= '';
END_IF

// Propagate Error to MoveRequest and State Machine
iMoveRequest.MoveRequestError(
    Error        := THIS^.bError,
    ErrorId      := THIS^.nErrorId,
    ErrorMessage := THIS^.sErrorMessage
);

iStateMachine.StateMachine(
    Error          := THIS^.bError, 
    InterlockEvent := THIS^.iInterlocks.Warning
);

// Brake and Status Mapping
iBrake.AxisState := iAxis.Status.eAxisState;

// Main Motion Status Structure
stMotionStatus.nMotionAxisID    := iAxis.Status.nAxisId;
stMotionStatus.bEnabled         := iInterlocks.PowerEnabled;
stMotionStatus.bHomeSensor      := iInterlocks.HomeSensor;
stMotionStatus.bLimitBwd        := iInterlocks.MoveBackwardEnabled;
stMotionStatus.bLimitFwd        := iInterlocks.MoveForwardEnabled;
stMotionStatus.fActDiff         := iAxis.Status.fMeasuredPositionDiff;
stMotionStatus.fActPosition     := iAxis.Status.fMeasuredPosition;
stMotionStatus.fActVelocity     := iAxis.Status.fMeasuredVelocity;
stMotionStatus.fOverride        := iAxis.Status.fPowerOverride;
stMotionStatus.bBusy            := iAxis.Status.bBusy;
stMotionStatus.bHomed           := iAxis.Status.bHomeDone;
stMotionStatus.bWarning         := iInterlocks.Warning;
stMotionStatus.bError           := THIS^.bError;
stMotionStatus.nErrorId         := THIS^.nErrorId;
stMotionStatus.sErrorMessage    := THIS^.sErrorMessage;

// Extended Motion Status (Debug, Testing)
stExMotionStatus.bMotionAxisError        := iAxis.Status.bError;
stExMotionStatus.nMotionAxisErrorId      := iAxis.Status.nErrorID;
stExMotionStatus.bInterlocksError        := iInterlocks.Error;
stExMotionStatus.nInterlocksError        := iInterlocks.ErrorID;
stExMotionStatus.eDriveState             := iStateMachine.MoveState;
stExMotionStatus.bAbortDone              := iAxis.Status.bAbortDone;
stExMotionStatus.bAborted                := iAxis.Status.bAborted;
stExMotionStatus.bLimHomeDone            := iAxis.Status.bLimHomeDone;
stExMotionStatus.bDriveWatchDogStatus    := iStateMachine.WatchDogStatus;
stExMotionStatus.bNewMoveReq             := iMoveRequest.Status.bNewMoveReq;
stExMotionStatus.bEnable                 := iMoveRequest.Status.bEnable;
stExMotionStatus.bIdling                 := iStateMachine.Idling;
stExMotionStatus.bExecute                := iMoveRequest.Status.bExecute;

METHOD PUBLIC CallAfterInit
VAR_INPUT
	stMotionCommand : REFERENCE TO ST_MotionCommand;
    stMotionStatus: REFERENCE TO ST_MotionStatus;
	stExMotionStatus : REFERENCE TO ST_ExtendedMotionStatus;
    iInterlocks : I_MotionInterlocks;
    iLogger : I_MotionLogger;
    iAxis: I_MotionAxis;
    iMoveRequest : I_MoveRequest;
    iStateMachine : I_StateMachine;
    iBrake : I_Brake;;
END_VAR
THIS^.iAxis := iAxis;
THIS^.iLogger:=iLogger;
THIS^.iBrake:=iBrake;
THIS^.iInterlocks:=iInterlocks;
THIS^.iMoveRequest :=iMoveRequest;
THIS^.iStateMachine := iStateMachine;
THIS^.stMotionCommand REF= stMotionCommand;
THIS^.stMotionStatus REF= stMotionStatus;
THIS^.stExMotionStatus REF= stExMotionStatus;
END_METHOD

//FB_Init is always available implicitly and it is used primarily for initialization.
//The return value is not evaluated. For a specific influence, you can also declare the
//methods explicitly and provide additional code there with the standard initialization
//code. You can evaluate the return value.
METHOD FB_Init: BOOL
VAR_INPUT
    bInitRetains: BOOL; // TRUE: the retain variables are initialized (reset warm / reset cold)
    bInCopyCode: BOOL;  // TRUE: the instance will be copied to the copy code afterward (online change)

	stMotionCommand : REFERENCE TO ST_MotionCommand;
    stMotionStatus: REFERENCE TO ST_MotionStatus;
	stExMotionStatus : REFERENCE TO ST_ExtendedMotionStatus;
    iInterlocks : I_MotionInterlocks;
    iLogger : I_MotionLogger;
    iAxis: I_MotionAxis;
    iMoveRequest : I_MoveRequest;
    iStateMachine : I_StateMachine;
    iBrake : I_Brake;
END_VAR
THIS^.iAxis := iAxis;
THIS^.iLogger:=iLogger;
THIS^.iBrake:=iBrake;
THIS^.iInterlocks:=iInterlocks;
THIS^.iMoveRequest :=iMoveRequest;
THIS^.iStateMachine := iStateMachine;
THIS^.stMotionCommand REF= stMotionCommand;
THIS^.stMotionStatus REF= stMotionStatus;
THIS^.stExMotionStatus REF= stExMotionStatus;
END_METHOD

PROPERTY SaveAxisParams : BOOL
SET
bSaveAxisParams := SaveAxisParams;
END_SET
END_PROPERTY

END_FUNCTION_BLOCK

// ---- POUs/FBs/Common/FB_MotionLogger.TcPOU
FUNCTION_BLOCK FB_MotionLogger IMPLEMENTS I_MotionLogger
VAR CONSTANT
    MOTION_LOGGER_MAX_MSGS_SIZE : UINT := 10;
END_VAR

VAR
	sName : STRING;
    nMaxMsg : UINT := MOTION_LOGGER_MAX_MSGS_SIZE; // configurable max log entries
    sLookedUpMsg :  MOTION_LOGGER_MSG;
    arLogMessages : ARRAY[1..MOTION_LOGGER_MAX_MSGS_SIZE] OF ST_MotionLogMessage;
    nLogWriteIdx : UINT := 1;
    nLogCount : UINT := 0;
    sLastMessage :  MOTION_LOGGER_MSG;
    {attribute 'pytmc' := '
        pv: PLC:sExtendedErrorMsgs
        io: i
        field: DESC Extended cyclic error message
    '}
    sExtendedErrorMsgs : STRING(1024);
END_VAR

METHOD PUBLIC CallAfterInit
VAR_INPUT
    sName : STRING; 
END_VAR
THIS^.sName := sName;
END_METHOD

METHOD Clear
VAR
    i : UINT;
END_VAR
FOR i := 1 TO nMaxMsg DO
    arLogMessages[i].sSource := '';
    arLogMessages[i].sMessage := '';
END_FOR
nLogWriteIdx := 1;
nLogCount := 0;
sLastMessage := '';
END_METHOD

METHOD ErrorCodeLookup : STRING
VAR_INPUT
	nErrorId	: UDINT;
END_VAR
CASE nErrorId OF
    // --- Common NC errors ---
    16#4221: sLookedUpMsg := 'Requested set velocity is not allowed';
    16#4222: sLookedUpMsg := 'Requested set position is not allowed';
    16#4223: sLookedUpMsg := 'No enable for controller and/or feed';
    16#4225: sLookedUpMsg := 'Drive not ready during axis start';
    16#4260: sLookedUpMsg := 'Drive disabled';
    16#42A0: sLookedUpMsg := 'Coupled axis error';
    16#4357: sLookedUpMsg := 'Negative limit hit';
    16#4358: sLookedUpMsg := 'Positive limit hit';
    16#4395: sLookedUpMsg := 'Set velocity not allowed';
    16#4466: sLookedUpMsg := 'Invalid I/O data for more than n continuous NC cycles (encoder)';
    16#4467: sLookedUpMsg := 'Encoder error: invalid actual position data';
    16#4550: sLookedUpMsg := 'Stall: position lag monitoring error';
    16#4650: sLookedUpMsg := 'Drive hardware not ready to operate';
    16#4655: sLookedUpMsg := 'Invalid IO data';
    16#4B07: sLookedUpMsg := 'Timeout axis function block after 6 seconds';
    16#4FFF: sLookedUpMsg := 'Unknown NC error (not in manual)';

    // --- Custom error definitions (make sure these enums are defined!) ---
    E_LCLSMotionError.ABORTED:   sLookedUpMsg := 'Aborted move request with active move in progress';
    E_LCLSMotionError.UNSAFE:    sLookedUpMsg := 'Position state unsafe';
    E_LCLSMotionError.INVALID:   sLookedUpMsg := 'Position state invalid';
    E_LCLSMotionError.TEST:      sLookedUpMsg := 'Fake testing error';

    // --- No error ---
    0:   sLookedUpMsg := '';
    
    // --- Fallback ---
    ELSE
        sLookedUpMsg := 'Contact PCDS to add new message';
END_CASE

ErrorCodeLookup := sLookedUpMsg;
END_METHOD

//FB_Init is always available implicitly and it is used primarily for initialization.
//The return value is not evaluated. For a specific influence, you can also declare the
//methods explicitly and provide additional code there with the standard initialization
//code. You can evaluate the return value.
METHOD FB_Init: BOOL
VAR_INPUT
    bInitRetains: BOOL; // TRUE: the retain variables are initialized (reset warm / reset cold)
    bInCopyCode: BOOL;  // TRUE: the instance will be copied to the copy code afterward (online change)  
    sName : STRING; 
END_VAR
THIS^.sName := sName;
END_METHOD

METHOD GetAllMessages : STRING(1024)
VAR
    i : UINT;
    idx : UINT;
END_VAR

VAR_OUTPUT

END_VAR
sExtendedErrorMsgs := '';
FOR i := 1 TO nLogCount DO
    //idx := (nLogWriteIdx + nLogCount - i - 1) MOD nMaxMsg + 1;
    sExtendedErrorMsgs := CONCAT(sExtendedErrorMsgs, '[');
    sExtendedErrorMsgs := CONCAT(sExtendedErrorMsgs, arLogMessages[i].sTimestamp);
    sExtendedErrorMsgs := CONCAT(sExtendedErrorMsgs, '] ');
    sExtendedErrorMsgs := CONCAT(sExtendedErrorMsgs, arLogMessages[i].sSource);
    sExtendedErrorMsgs := CONCAT(sExtendedErrorMsgs, ' ');
    sExtendedErrorMsgs := CONCAT(sExtendedErrorMsgs, TO_STRING(arLogMessages[i].eLevel));
    sExtendedErrorMsgs := CONCAT(sExtendedErrorMsgs, ': ');
    sExtendedErrorMsgs := CONCAT(sExtendedErrorMsgs, arLogMessages[i].sMessage);
    sExtendedErrorMsgs := CONCAT(sExtendedErrorMsgs, '\n');
END_FOR
GetAllMessages := sExtendedErrorMsgs;
END_METHOD

METHOD GetMessageCount : UINT
VAR_OUTPUT
    nCount : UINT;
END_VAR
nCount := nLogCount;
END_METHOD

METHOD Logger
VAR_INPUT
    Message : STRING;
    Level   : E_MotionLogLevel := E_MotionLogLevel.INFO;
    Source  : STRING := '';
END_VAR

VAR
	fbTimeStamp   : FB_LocalSystemTime := ( bEnable := TRUE, dwCycle := 1 );
    logMessage : ST_MotionLogMessage;
END_VAR
// Prepare record
logMessage.sSource     := CONCAT(sName, CONCAT(':', Source));
logMessage.sMessage    := Message;
logMessage.eLevel      := Level;

// Get timestamp; use SYSTEMTIME, DT, or T_TIMESTAMP depending on platform
fbTimeStamp();
logMessage.sTimestamp :=SYSTEMTIME_TO_STRING(fbTimeStamp.systemTime); // Or alternative if not available

// Save to buffer
arLogMessages[nLogWriteIdx] := logMessage;
sLastMessage := Message;

// Rotate buffer
nLogWriteIdx := nLogWriteIdx + 1;
IF nLogWriteIdx > nMaxMsg THEN
    nLogWriteIdx := 1;
END_IF
IF nLogCount < nMaxMsg THEN
    nLogCount := nLogCount + 1;
END_IF
END_METHOD

{warning 'Add property implementation'}
PROPERTY Name : STRING
GET
END_GET
END_PROPERTY

END_FUNCTION_BLOCK

// ---- POUs/FBs/Containers/FB_MotionStageNC.TcPOU
{attribute 'call_after_init'}
FUNCTION_BLOCK FB_MotionStageNC IMPLEMENTS I_MotionStage
VAR

    {attribute 'no_copy'}
    AxisRef : REFERENCE TO AXIS_REF;
   {attribute 'pytmc' := 'pv:'}
    stMotionCommand : ST_MotionCommand;
    // Misc axis status information for the IOC
    {attribute 'pytmc' := '
        pv: PLC:AxisStatus
        io: i
        field: DESC Axis motion status.
    '}
    stMotionStatus: ST_MotionStatus;
   {attribute 'hide'}
   {attribute 'pytmc' := 'pv:'}
	stExMotionStatus : ST_ExtendedMotionStatus;
   {attribute 'hide'}
    iPersistentDataStorage : I_PersistentDataStorage;
    fbMotionLogger : FB_MotionLogger(sName := sName);
    //Brakes : brake fb participate in sync comm with fbMotionDrive, fbMotionAxis and fbMotionInterlocks
    fbBrake : FB_BrakeNC := (BrakeMode := E_StageBrakeMode.IF_MOVING);
    // common interlocks
	{attribute 'pytmc' := 'pv:'}
    fbMotionInterlocksCommon : FB_MotionInterlocksCommon(
		iMotionLogger := fbMotionLogger, 
	);
    // stage with Limit switches
    fbLimSwStatus : FB_LimSwStatus();
	
    fbMotionInterlocksLimSw : FB_MotionInterlocksLimSw ( 
		iMotionInterlocksCommon:=fbMotionInterlocksCommon, 
		iLimSwStatus:=fbLimSwStatus,
		iMotionLogger := fbMotionLogger
	);
	
	fbHome : FB_HomeNC(
        AxisRef := AxisRef,
        iMotionLogger := fbMotionLogger,
        iLimSwStatus := fbLimSwStatus
    );

    fbHalt : FB_HaltNC(
		AxisRef := AxisRef,
		iMotionLogger := fbMotionLogger
	);
	
    fbPower : FB_PowerNC(
		AxisRef := AxisRef,
		iMotionLogger := fbMotionLogger
	);
	
    fbReset : FB_ResetNC(
		AxisRef := AxisRef,
		iMotionLogger := fbMotionLogger
	);
	
    fbMoveAbsolute : FB_MoveAbsoluteNC(
		AxisRef := AxisRef,
		iMotionLogger := fbMotionLogger
	);
	
    {attribute 'pytmc' := 'pv:'}
    fbReadParameter : FB_ReadParameterNC(
		AxisRef := AxisRef,
		iMotionLogger := fbMotionLogger
	);
    fbWriteParameter : FB_WriteParameterNC(
		AxisRef := AxisRef, 
		iMotionLogger := fbMotionLogger
	);
	
    fbParamsSaveRestore : FB_ParamsSaveRestoreNC(
        AxisRef := AxisRef,
        iPersistentDataStorage := iPersistentDataStorage,
		iMotionLogger := fbMotionLogger
    );

    {attribute 'pytmc' := 'pv:'}
    fbEncoderScaling : FB_EncoderScaling();

    {attribute 'pytmc' := 'pv:'}
    fbBacklashCompensation : FB_BacklashCompensationNC(
		AxisRef := AxisRef, 
		iMotionLogger := fbMotionLogger
	);
	
	{attribute 'pytmc' := 'pv:'}
    fbMotionAxis : FB_MotionAxisNC(
		AxisRef := AxisRef,
		iMotionLogger := fbMotionLogger,
        iHome := fbHome,
        iHalt := fbHalt,
        iPower := fbPower,
        iReset := fbReset,
        iMoveAbsolute := fbMoveAbsolute,
        iReadParameter := fbReadParameter,
        iWriteParameter  := fbWriteParameter,
        iParamsSaveRestore:= fbParamsSaveRestore,
        iEncoderScaling := fbEncoderScaling,
        iBacklashCompensation :=fbBacklashCompensation,
    );
		// Motion Requests
	{attribute 'pytmc' := 'pv:'}
    fbMoveRequest : FB_EpicsMoveRequest(
		stMotionCommand:=stMotionCommand,
		stMotionStatus:=stMotionStatus
	);

    fbStateMachine  : FB_MotionDriveStateMachine(
		    stMotionCommand:=stMotionCommand,
            iMotionAxis:=fbMotionAxis,
            iMoveRequest:=fbMoveRequest,
			iMotionLogger := fbMotionLogger
    );
	
	fbMotionDrive : FB_MotionDrive(	
		stMotionCommand :=stMotionCommand,
		stMotionStatus:=stMotionStatus,
		stExMotionStatus :=stExMotionStatus,
		iInterlocks :=fbMotionInterlocksLimSw,
		iLogger :=fbMotionLogger,
		iAxis:=fbMotionAxis,
		iMoveRequest :=fbMoveRequest,
		iStateMachine :=fbStateMachine,
		iBrake :=fbBrake
	);
    // Name to use for log messages, fast faults, etc.
    {attribute 'hide'}
    sName : T_MaxString;
	bSaveAxisParams : BOOL;
END_VAR

// 1. Update all hardware IO/limit/interlock state at the very start
    fbLimSwStatus();
    fbMotionInterlocksCommon();
    fbMotionInterlocksLimSw();

    // 2. Call move request arbitration block (process user/sequencer requests)
    fbMoveRequest();

    // 3. Call orchestration: requests, coordination, error logic (must come BEFORE NC blocks)
    fbMotionDrive();

    // 4. All NC-level and axis control function blocks (must be called EVERY scan)
    fbReset();
    fbHalt();
    fbPower();
    fbBacklashCompensation();
    fbMoveAbsolute();
    fbHome();
    fbReadParameter();
    fbWriteParameter();
    fbParamsSaveRestore();
    fbEncoderScaling();
    fbMotionAxis();

    // 5. State machine/coordination logic using up-to-date status after NC block execution
    fbStateMachine();

    // 6. Brake and any final safety logic
    fbBrake();
	
	//7. 
	fbMotionLogger();

METHOD AbsoluteMove
VAR_INPUT
	Position :LREAL;
	Velocity :LREAL;
	Acceleration :LREAL;
	Deceleration :LREAL;
END_VAR
stMotionCommand.fPosition := Position;
stMotionCommand.fVelocity := Velocity;
stMotionCommand.fAcceleration := Acceleration;
stMotionCommand.fDeceleration := Deceleration;
stMotionCommand.fDeceleration := Deceleration;
stMotionCommand.bMoveCmd := TRUE;
//stMotionInterface.bExecute:=TRUE;
END_METHOD

{warning 'Add method implementation '}
METHOD AbsoluteMoveWithBacklashCompensation
VAR_INPUT
	Position	: LREAL;
	Velocity	: LREAL;
	Acceleration	: LREAL;
	Deceleration	: LREAL;
END_VAR
 AbsoluteMove(	
	Position	:= Position,
	Velocity	:= Velocity,
	Acceleration	:= Acceleration,
	Deceleration	:= Deceleration
);
//fbBacklashCompensation.BacklashCompensation(Enable := TRUE, RampVelo := Velocity/10.0);
END_METHOD

{attribute 'call_after_init'}
METHOD PRIVATE CallAfterInit
fbMotionInterlocksCommon.CallAfterInit(
	iMotionLogger := THIS^.fbMotionLogger, 
);
//fbLimSwStatus.CallAfterInit(iMotionLogger := THIS^.fbMotionLogger);
fbMotionInterlocksLimSw.CallAfterInit(
	iMotionInterlocksCommon := THIS^.fbMotionInterlocksCommon,
	iLimSwStatus := THIS^.fbLimSwStatus,
	iMotionLogger := THIS^.fbMotionLogger
);

// Pass correctly initialized Motion axis dependencies
fbHome.CallAfterInit(
        AxisRef := THIS^.AxisRef,
        iMotionLogger := THIS^.fbMotionLogger,
        iLimSwStatus := THIS^.fbLimSwStatus
);

fbHalt.CallAfterInit(
	AxisRef := THIS^.AxisRef,
	iMotionLogger := THIS^.fbMotionLogger
);

fbPower.CallAfterInit(
	AxisRef := THIS^.AxisRef,
	iMotionLogger := THIS^.fbMotionLogger
);

fbReset.CallAfterInit(
	AxisRef := THIS^.AxisRef,
	iMotionLogger := THIS^.fbMotionLogger
);

fbMoveAbsolute.CallAfterInit(
	AxisRef := THIS^.AxisRef,
	iMotionLogger := THIS^.fbMotionLogger
);

fbReadParameter.CallAfterInit(
	AxisRef := THIS^.AxisRef,
	iMotionLogger := THIS^.fbMotionLogger
);

fbWriteParameter.CallAfterInit(
	AxisRef := THIS^.AxisRef,
	iMotionLogger := THIS^.fbMotionLogger
);

fbParamsSaveRestore.CallAfterInit(
	AxisRef := THIS^.AxisRef,
	iPersistentDataStorage := THIS^.iPersistentDataStorage,
	iMotionLogger := THIS^.fbMotionLogger
);

fbBacklashCompensation.CallAfterInit(
	AxisRef := THIS^.AxisRef,
	iMotionLogger := THIS^.fbMotionLogger
);

fbMotionAxis.CallAfterInit(
	AxisRef := THIS^.AxisRef,
	iMotionLogger := THIS^.fbMotionLogger,
    iHome := THIS^.fbHome,
    iHalt := THIS^.fbHalt,
    iPower := THIS^.fbPower,
    iReset := THIS^.fbReset,
    iMoveAbsolute := THIS^.fbMoveAbsolute,
    iReadParameter := THIS^.fbReadParameter,
    iWriteParameter  := THIS^.fbWriteParameter,
    iParamsSaveRestore:= THIS^.fbParamsSaveRestore,
    iEncoderScaling := THIS^.fbEncoderScaling,
    iBacklashCompensation := THIS^.fbBacklashCompensation
);


fbMoveRequest.CallAfterInit(
	stMotionCommand:= THIS^.stMotionCommand,
	stMotionStatus:= THIS^.stMotionStatus
);

fbMotionDrive.CallAfterInit(	
	stMotionCommand :=THIS^.stMotionCommand,
	stMotionStatus:=THIS^.stMotionStatus,
	stExMotionStatus :=THIS^.stExMotionStatus,
	iInterlocks :=THIS^.fbMotionInterlocksLimSw,
	iLogger :=THIS^.fbMotionLogger,
	iAxis:=THIS^.fbMotionAxis,
	iMoveRequest :=THIS^.fbMoveRequest,
	iStateMachine :=THIS^.fbStateMachine,
	iBrake :=THIS^.fbBrake
);
	
fbStateMachine.CallAfterInit(
	iMotionAxis:=THIS^.fbMotionAxis, 
	iMoveRequest:=THIS^.fbMoveRequest, 
	stMotionCommand:=THIS^.stMotionCommand,
	iMotionLogger := THIS^.fbMotionLogger
);
END_METHOD

METHOD INTERNAL EnableBacklashCompensation
VAR_INPUT
    UserEnable : BOOL;
    Compensation : LREAL;
END_VAR
THIS^.fbMotionAxis.EnableBacklashCompensation(UserEnable:=UserEnable, Compensation:=Compensation);
END_METHOD

METHOD INTERNAL EnableInterlocks : BOOL
VAR_INPUT
END_VAR
THIS^.fbMotionInterlocksCommon.EnableInterlocks(
	UserEnable:=TRUE, 
	HardwareEnable:=TRUE
);
END_METHOD

METHOD INTERNAL EnableLimits
VAR_INPUT
	ForwardEnable : BOOL;
	BackwardEnable : BOOL;
	HomeEnable : BOOL;
END_VAR
fbLimSwStatus.LimitBackwardEnable := BackwardEnable;
fbLimSwStatus.LimitForwardEnable:=ForwardEnable;
fbLimSwStatus.LimitHome := HomeEnable ;
END_METHOD

PROPERTY ExMotionStatus : REFERENCE TO ST_ExtendedMotionStatus
GET
ExMotionStatus REF= stExMotionStatus;
END_GET
END_PROPERTY

//FB_Init is always available implicitly and it is used primarily for initialization.
//The return value is not evaluated. For a specific influence, you can also declare the
//methods explicitly and provide additional code there with the standard initialization
//code. You can evaluate the return value.
METHOD FB_Init: BOOL
VAR_INPUT
    bInitRetains: BOOL; // TRUE: the retain variables are initialized (reset warm / reset cold)
    bInCopyCode: BOOL;  // TRUE: the instance will be copied to the copy code afterward (online change)
    AxisRef : REFERENCE TO AXIS_REF;
    iPersistentDataStorage : I_PersistentDataStorage;
    sName : T_MaxString;
END_VAR
THIS^.AxisRef REF= AxisRef;
THIS^.iPersistentDataStorage := iPersistentDataStorage;
THIS^.sName := sName;
END_METHOD

METHOD Halt
THIS^.stMotionCommand.bHalt := TRUE;
END_METHOD

METHOD Home
VAR_INPUT
	HomePosition	: LREAL;
	HomeMode	: INT;
END_VAR
THIS^.stMotionCommand.fHomePosition := HomePosition;
THIS^.stMotionCommand.nCmdData := HomeMode;
THIS^.stMotionCommand.bHomeCmd := TRUE;
END_METHOD

PROPERTY MotionCmd : REFERENCE TO ST_MotionCommand
GET
MotionCmd REF= stMotionCommand;
END_GET
END_PROPERTY

{warning 'Add property implementation'}
PROPERTY MotionStatus : REFERENCE TO ST_MotionStatus
GET
MotionStatus REF= stMotionStatus;
END_GET
END_PROPERTY

{warning 'Add method implementation '}
METHOD Reset
stMotionCommand.bReset:=TRUE;
END_METHOD

PROPERTY SaveAxisParams : BOOL
SET
THIS^.fbMotionDrive.SaveAxisParams := bSaveAxisParams;
END_SET
END_PROPERTY

METHOD INTERNAL SetModeEnableLimits
VAR_INPUT  
	LimBackward : BOOL; 
	LimForward: BOOL; 
	BrakeMode : E_StageBrakeMode; 
	EnableMode: ENUM_StageEnableMode; 
	HomeMode: E_EpicsHomeCmd;
END_VAR
END_METHOD

METHOD StateMove
VAR_INPUT
	Execute : BOOL;
END_VAR
stMotionCommand.bMoveCmd := Execute;
END_METHOD

METHOD INTERNAL UpdateInterlockUserEnable
VAR_INPUT
	UserEnable : BOOL;
	HardwareEnable : BOOL;
END_VAR
fbMotionInterlocksCommon.EnableInterlocks(
	UserEnable:=UserEnable,
	HardwareEnable:=HardwareEnable
);
END_METHOD

END_FUNCTION_BLOCK

// ---- POUs/FBs/NC/FB_ParamsSaveRestoreNC.TcPOU
FUNCTION_BLOCK FB_ParamsSaveRestoreNC IMPLEMENTS I_ParamsSaveRestore
VAR
    {attribute 'no_copy'}
    AxisRef : REFERENCE TO AXIS_REF;
    {attribute 'hide'}
    iPersistentDataStorage : I_PersistentDataStorage := 0;
	iMotionLogger : I_MotionLogger := 0;
    // save and restore
    {attribute 'hide'}
    fbSetPos: MC_SetPosition;
    {attribute 'hide'}
    bClearPositionLag : BOOL := TRUE;
    {attribute 'hide'}
    nLatchErrId : BOOL;
    {attribute 'hide'}
    bRestoreDone 	: BOOL;
    {attribute 'hide'}
    bRestoreError 	: BOOL;
    {attribute 'hide'}
    nRestoreErrorID : UDINT;
    {attribute 'hide'}
    // save and Restore
    RestoreTimer: TON;
    {attribute 'hide'}
    bRestoreInit: BOOL;
    {attribute 'hide'}
    bRestoreLoad: BOOL;
    {attribute 'hide'}
    nLatchError: UDINT;
    {attribute 'hide'}
    bEncError: BOOL;
    {attribute 'hide'}
    tRetryDelay: TIME := T#1S;
    {attribute 'hide'}
    tRefreshDelay: TIME := T#1S;
    {attribute 'hide'}
    bUpdateEnable : BOOL;
    {attribute 'hide'}
    bExecute : BOOL;
    {attribute 'hide'}
    nMaxRetries: UINT := 10;
    {attribute 'hide'}
    nCurrTries: UINT := 0;
    {attribute 'hide'}
    bRestoreWaitRetry: BOOL;
    {attribute 'hide'}
    tonRestoreRetry: TON;
    {attribute 'hide'}
    tRefreshTime : TIME := T#1S;
    {attribute 'hide'}
    bError				: BOOL;
    {attribute 'hide'}
    nErrorId			: UDINT:=0;
    {attribute 'hide'}
    sMessage : T_MAXSTRING;
    {attribute 'hide'}
    bSaveEnabled	: BOOL := TRUE;
    {attribute 'hide'}
    bDone : BOOL;
    {attribute 'hide'}
    bBusy    : BOOL;
END_VAR

VAR PERSISTENT
    {attribute 'conditionalshow'}
    bSaved: BOOL;
    {attribute 'conditionalshow'}
    fSavedPosition: LREAL;
END_VAR

IF NOT __ISVALIDREF(AxisRef) THEN
    RETURN;
END_IF

AxisRef.ReadStatus();

RestoreAxisParams();

// Save Encoder position
// needs some pre-conditions to use persistent storage
IF bSaveEnabled THEN
    // Check ST_MotionStage for an encoder error (range 0x44nn)
    bEncError:= AxisRef.Status.Error AND  ( AxisRef.Status.ErrorID  >= 16#4400  AND AxisRef.Status.ErrorID <= 16#44FF );
    // Do not save if we're currently loading or if there is an encoder error
    IF NOT bRestoreLoad AND NOT bEncError AND NOT bRestoreWaitRetry THEN
        fSavedPosition := AxisRef.NcToPlc.ActPos;
        // This persistent variable lets us check if anything was saved
        // It will be TRUE at startup if we have saved values
        bSaved := TRUE;
        (*
            use this with a timer of a change threshold on the fActPosition
            to trigger a save from this PLC program. otherwise this will be a spamming
            persistence, filling up the disk.
        *)
        //iPersistentDataStorage.TriggerWriteOfPersistentData := bSaveEnabled;
    END_IF
END_IF

PROPERTY Busy : BOOL
GET
Busy := bBusy;
END_GET
END_PROPERTY

METHOD PUBLIC CallAfterInit
VAR_INPUT
    AxisRef : REFERENCE TO AXIS_REF;
    iPersistentDataStorage : I_PersistentDataStorage;
	iMotionLogger : I_MotionLogger;
END_VAR
THIS^.AxisRef REF= AxisRef;
THIS^.iPersistentDataStorage := iPersistentDataStorage;
THIS^.iMotionLogger := iMotionLogger;
END_METHOD

PROPERTY Done : BOOL
GET
Done := bRestoreDone;
END_GET
END_PROPERTY

PROPERTY Error : BOOL
GET
Error := bError;
END_GET
END_PROPERTY

PROPERTY ErrorID : UDINT
GET
ErrorID := nErrorID;
END_GET
END_PROPERTY

//FB_Init is always available implicitly and it is used primarily for initialization.
//The return value is not evaluated. For a specific influence, you can also declare the
//methods explicitly and provide additional code there with the standard initialization
//code. You can evaluate the return value.
METHOD FB_Init: BOOL
VAR_INPUT
    bInitRetains: BOOL; // TRUE: the retain variables are initialized (reset warm / reset cold)
    bInCopyCode: BOOL;  // TRUE: the instance will be copied to the copy code afterward (online change)
    AxisRef : REFERENCE TO AXIS_REF;
    iPersistentDataStorage : I_PersistentDataStorage;
	iMotionLogger : I_MotionLogger;
END_VAR
THIS^.AxisRef REF= AxisRef;
THIS^.iPersistentDataStorage := iPersistentDataStorage;
THIS^.iMotionLogger := iMotionLogger;
END_METHOD

PROPERTY Message : T_MAXSTRING
GET
Message := sMessage;
END_GET
END_PROPERTY

METHOD RestoreAxisParams
// Trigger a load if anything was saved at all
IF NOT bRestoreInit THEN
    bRestoreInit := TRUE;
    bRestoreLoad S= bSaved;
    fbSetPos.Options.ClearPositionLag := TRUE;
END_IF

// Set our position if bRestoreLoad is true
fbSetPos( Axis:=AxisRef, Execute:=bRestoreLoad, Position:=fSavedPosition);

// Only load once, at startup
bRestoreLoad R= fbSetPos.Done OR fbSetPos.Error;

IF fbSetPos.Error THEN
    // Keep the error latched, it can disappear if Execute is set to FALSE
    nLatchError := fbSetPos.ErrorID;
    nCurrTries := nCurrTries + 1;
    IF nCurrTries >= nMaxRetries THEN
        // Alert the user that something has gone wrong
        bError := TRUE;
        nErrorId := nLatchError;
        sMessage := 'Error loading previously saved position.';
    ELSE
        // Reset the FB for the next retry
        fbSetPos( Axis:=THIS^.AxisRef, Execute:=bRestoreLoad, Position:=fSavedPosition);
        // Try again
        bRestoreWaitRetry := TRUE;
    END_IF
ELSE
    bRestoreDone := TRUE;
END_IF

tonRestoreRetry( IN := bRestoreWaitRetry, PT := tRetryDelay);
bRestoreLoad S= tonRestoreRetry.Q;
bRestoreWaitRetry R= tonRestoreRetry.Q;
END_METHOD

METHOD SaveAxisParams
VAR_INPUT
    Enable	: BOOL;
END_VAR
THIS^.bSaveEnabled := Enable;
END_METHOD

PROPERTY SavedPosition : LREAL
GET
SavedPosition := fSavedPosition;
END_GET
END_PROPERTY

END_FUNCTION_BLOCK

// ---- Test/Containers/FB_MotionStageNC_Test.TcPOU
FUNCTION_BLOCK INTERNAL FB_MotionStageNC_Test EXTENDS FB_TestSuite
VAR
    fbPersistentDataStorage :  ARRAY[1..17] OF FB_PersistentDataStorage;
 	fbAxisRef :   ARRAY[1..17] OF AXIS_REF;
END_VAR

GivenMoveCmdAndMoveOkIfResetThenAbortMove_Test1();
GivenMoveCmdAndMoveOkIfHaltThenAbortMove_Test2();
GivenMoveCmdAndMoveOkMoveToTarget1ThenTarget2_Test3();
GivenMoveCmdAndValidInterlocksThenMoveToTarget_Test4();
GivenMoveCmdValidInterlockAndWrongMotionParamsThenGotoErrorStateIfResetThenGotoInitState_Test5();
GivenMoveCmdAndMoveOkAndPositiveBacklashEnabledThenMoveToTargetWithCompensation_Test6();
GivenMoveCmdAndMoveOkAndNegativeBacklashEnabledThenMoveToTargetWithCompensation_Test7();
GivenHomeCmdAndAbsoluteSetAndMoveOkThenMoveToUserDefinedHomePosition_Test8();
GivenHomeCmdNoneAndMoveOkThenSetHomeFlag_Test9();
GivenHomeCmdLowLimitModeBackwardSwPulseMoveOkThenMoveToUserDefinedHomePosition_Test10();
GivenHomeCmdHighLimitModeForwardSwPulseMoveOkThenMoveToUserDefinedHomePosition_Test11();
GivenHomeCmdHomeViaLowModeHomeSwPulseMoveOkThenMoveToUserDefinedHomePosition_Test12();
GivenHomeCmdHomeViaHighModeHomeSwPulseMoveOkThenMoveToUserDefinedHomePosition_Test13();
GivenHomeCmdHomeViaHighModeForwardSwPulseBeforeHomeSwPulseThenMoveToUserDefinePosition_Test14();
GivenHomeCmdHomeViaLowModeBackwardSwPulseBeforeHomeSwPulseThenMoveToUserDefinePosition_Test15();
GivenHomeCmdLowLimitModeAndResetThenAbortHoming_Test16();
OverallStageFeaturesAndOperationalTests_Test17();

METHOD PRIVATE GivenHomeCmdAndAbsoluteSetAndMoveOkThenMoveToUserDefinedHomePosition_Test8
VAR_INST
   fbMotionStage : FB_MotionStageNC(	sName := 'Test8',
                                        AxisRef := fbAxisRef[8],
                                        iPersistentDataStorage := fbPersistentDataStorage[8]
                                    ) :=(SaveAxisParams := FALSE);
									
    fbTestTimer: TON := (IN:=TRUE, PT:=T#10S);
    nTestStep : INT;
END_VAR
TEST(__POUNAME());


CASE nTestStep OF
    0:
			// Enable safety interlocks and hardware limits
        fbMotionStage.EnableLimits(
			BackwardEnable:=TRUE, 
			ForwardEnable:=TRUE,
			HomeEnable:=FALSE
		);
        fbMotionStage.EnableInterlocks();
		nTestStep := 1;
	1:
		fbMotionStage.Home(HomePosition:=20.0, HomeMode:=E_EPicsHomeCmd.ABSOLUTE_SET);
		nTestStep := 2;
	2:
		IF fbMotionStage.stMotionStatus.bDone THEN
			AssertTrue(Condition :=(fbMotionStage.stMotionCommand.fHomePosition - fbAxisRef[8].NcToPlc.ActPos) = 0, Message := 'Hone position not set #1');
			nTestStep := 3;
		END_IF	
END_CASE

fbTestTimer();
fbMotionStage();

IF nTestStep = 3 THEN

TEST_FINISHED();
ELSIF fbTestTimer.Q THEN
    AssertTrue(
        Condition := FALSE,
        Message := CONCAT('Timed out at step: ', TO_STRING(nTestStep))
    );
    TEST_FINISHED();
END_IF
END_METHOD

METHOD PRIVATE GivenHomeCmdHighLimitModeForwardSwPulseMoveOkThenMoveToUserDefinedHomePosition_Test11
VAR_INST
   fbMotionStage : FB_MotionStageNC(	sName := 'Test11',
                                        AxisRef := fbAxisRef[11],
                                        iPersistentDataStorage := fbPersistentDataStorage[11]
                                    ) :=(SaveAxisParams := FALSE);
									
    fbTestTimer: TON := (IN:=TRUE, PT:=T#10S);
    fbCamSwitchPulserSearch: TON := (IN:=TRUE, PT:=T#500MS);
    fbCamSwitchPulserSync: TON := (PT:=T#1000MS);
    nTestStep : INT;
END_VAR
TEST(__POUNAME());

CASE nTestStep OF
    0: // Enable all interlocks/limits to be ready for homing
        fbMotionStage.EnableLimits(
			BackwardEnable:=TRUE, 
			ForwardEnable:=TRUE,
			HomeEnable:=FALSE
		);
        fbMotionStage.EnableInterlocks();
        nTestStep := 1;

    1: // Issue home command (to low limit)
        fbMotionStage.Home(HomePosition := 20.0, HomeMode := E_EpicsHomeCmd.HIGH_LIMIT);
        nTestStep := 2;

    2: // Simulate limit switch drop/restore with cam switch events
        IF fbCamSwitchPulserSearch.Q THEN
			// simulate limit release
			fbMotionStage.EnableLimits(
				BackwardEnable:=TRUE, 
				ForwardEnable:=FALSE,
				HomeEnable:=FALSE
			);
            fbCamSwitchPulserSearch.IN := FALSE;
            fbCamSwitchPulserSync.IN := TRUE;
            nTestStep := 3;
        END_IF

    3: // Restore limit after cam event
        IF fbCamSwitchPulserSync.Q THEN
			fbMotionStage.EnableLimits(
				BackwardEnable:=TRUE, 
				ForwardEnable:=TRUE,
				HomeEnable:=FALSE
			);
            nTestStep := 4;
        END_IF

    4: // Wait for home sequence completion
        IF fbMotionStage.stMotionStatus.bDone THEN
            nTestStep := 5;
        END_IF
END_CASE

fbCamSwitchPulserSearch();
fbCamSwitchPulserSync();
fbTestTimer();
fbMotionStage();

IF nTestStep = 5 THEN
    AssertTrue(
        Condition := fbAxisRef[11].Status.Homed,
        Message := 'Axis not calibrated #1'
    );
    AssertEquals_LREAL(
        Delta := 0.001,
        Expected := fbMotionStage.stMotionCommand.fHomePosition,
        Actual := fbAxisRef[11].NcToPlc.ActPos,
        Message := 'Position is not the expected #2'
    );
    TEST_FINISHED();
ELSIF fbTestTimer.Q THEN
    AssertTrue(
        Condition := FALSE,
        Message := CONCAT('Timed out at step: ', TO_STRING(nTestStep))
    );
    TEST_FINISHED();
END_IF
END_METHOD

METHOD PRIVATE GivenHomeCmdHomeViaHighModeForwardSwPulseBeforeHomeSwPulseThenMoveToUserDefinePosition_Test14
VAR_INST
   fbMotionStage : FB_MotionStageNC(	sName := 'Test14',
                                        AxisRef := fbAxisRef[14],
                                        iPersistentDataStorage := fbPersistentDataStorage[14]
                                    ) :=(SaveAxisParams := FALSE);
									
    fbTestTimer: TON := (IN:=TRUE, PT:=T#10S);
    fbCamSwitchPulserSearch: TON := (IN:=TRUE, PT:=T#500MS);
    fbCamSwitchPulserSync: TON := (PT:=T#1000MS);
    nTestStep : INT;
END_VAR
TEST(__POUNAME());

CASE nTestStep OF
    0: // Enable all interlocks/limits for initial homing (home switch not active yet!)
        fbMotionStage.EnableLimits(
            BackwardEnable := TRUE, 
            ForwardEnable  := TRUE,
            HomeEnable     := FALSE
        );
        fbMotionStage.EnableInterlocks();
        nTestStep := 1;

    1: // Issue homing command (via high limit, should travel to positive end first)
        fbMotionStage.Home(
            HomePosition := 5.0,
            HomeMode := E_EpicsHomeCmd.HOME_VIA_HIGH
        );
        nTestStep := 2;

    2: // Simulate forward limit drop
        IF fbCamSwitchPulserSearch.Q THEN
            fbMotionStage.EnableLimits(
                BackwardEnable := TRUE, 
                ForwardEnable  := FALSE,
                HomeEnable     := FALSE
            );
            fbCamSwitchPulserSearch.IN := FALSE;
            fbCamSwitchPulserSync.IN := TRUE;
            nTestStep := 3;
        END_IF

    3: // Restore forward limit after event
        IF fbCamSwitchPulserSync.Q THEN
            fbMotionStage.EnableLimits(
                BackwardEnable := TRUE, 
                ForwardEnable  := TRUE,
                HomeEnable     := FALSE
            );
            fbCamSwitchPulserSync.IN := FALSE;
            nTestStep := 4;
        END_IF

    4: // Wait for "first stage" (positive limit) homing done (i.e. LimHomeDone signals)
        IF fbMotionStage.stExMotionStatus.bLimHomeDone THEN
            // prepare for home switch pulse
            fbCamSwitchPulserSearch.IN := TRUE;
            fbCamSwitchPulserSync.IN := FALSE;
            nTestStep := 5;
        END_IF

    5: // Simulate home switch engagement (simulate HomeEnable = TRUE)
        IF fbCamSwitchPulserSearch.Q THEN
            fbMotionStage.EnableLimits(
                BackwardEnable := TRUE, 
                ForwardEnable  := TRUE,
                HomeEnable     := TRUE
            );
            fbCamSwitchPulserSearch.IN := FALSE;
            fbCamSwitchPulserSync.IN := TRUE;
            nTestStep := 6;
        END_IF

    6: // Simulate home switch disengagement (return HomeEnable to FALSE)
        IF fbCamSwitchPulserSync.Q THEN
            fbMotionStage.EnableLimits(
                BackwardEnable := TRUE, 
                ForwardEnable  := TRUE,
                HomeEnable     := FALSE
            );
            fbCamSwitchPulserSync.IN := FALSE;
            nTestStep := 7;
        END_IF 

    7: // Wait for overall homing to complete (done)
        IF fbMotionStage.stMotionStatus.bDone THEN
            nTestStep := 8;
        END_IF
END_CASE

// Cyclic calls required for timer and cam events and motion stage
fbCamSwitchPulserSearch();
fbCamSwitchPulserSync();
fbTestTimer();
fbMotionStage();

IF nTestStep = 8 THEN
    AssertTrue(
        Condition := fbAxisRef[14].Status.Homed,
        Message := 'Axis not calibrated #1'
    );
    AssertEquals_LREAL(
        Delta := 0.001,
        Expected := fbMotionStage.stMotionCommand.fHomePosition,
        Actual := fbAxisRef[14].NcToPlc.ActPos,
        Message := 'Position is not the expected #2'
    );
    TEST_FINISHED();
ELSIF fbTestTimer.Q THEN
    AssertTrue(
        Condition := FALSE,
        Message := CONCAT('Timed out at step: ', TO_STRING(nTestStep))
    );
    TEST_FINISHED();
END_IF
END_METHOD

METHOD PRIVATE GivenHomeCmdHomeViaHighModeHomeSwPulseMoveOkThenMoveToUserDefinedHomePosition_Test13
VAR_INST
   fbMotionStage : FB_MotionStageNC(	sName := 'Test13',
                                        AxisRef := fbAxisRef[13],
                                        iPersistentDataStorage := fbPersistentDataStorage[13]
                                    ):=(SaveAxisParams := FALSE);
									
    fbTestTimer: TON := (IN:=TRUE, PT:=T#10S);
    fbCamSwitchPulserSearch: TON := (IN:=TRUE, PT:=T#500MS);
    fbCamSwitchPulserSync: TON := (PT:=T#1000MS);
    nTestStep : INT;
END_VAR
TEST(__POUNAME());

CASE nTestStep OF
    0: // Enable all interlocks/limits to be ready for homing
		fbMotionStage.EnableLimits(
			BackwardEnable:=TRUE, 
			ForwardEnable:=TRUE,
			HomeEnable:=FALSE
		);
        fbMotionStage.EnableInterlocks();
        nTestStep := 1;

    1: // Issue home command (to low limit)
        fbMotionStage.Home(HomePosition := 20.0, HomeMode := E_EpicsHomeCmd.HOME_VIA_HIGH);
        nTestStep := 2;

    2: // Simulate limit switch drop/restore with cam switch events
        IF fbCamSwitchPulserSearch.Q THEN
			fbMotionStage.EnableLimits(
				BackwardEnable:=TRUE, 
				ForwardEnable:=TRUE,
				HomeEnable:=TRUE
			);
            fbCamSwitchPulserSearch.IN := FALSE;
            fbCamSwitchPulserSync.IN := TRUE;
            nTestStep := 3;
        END_IF

    3: // Restore limit after cam event
        IF fbCamSwitchPulserSync.Q THEN
			fbMotionStage.EnableLimits(
				BackwardEnable:=TRUE, 
				ForwardEnable:=TRUE,
				HomeEnable:=FALSE
			);
            nTestStep := 4;
        END_IF

    4: // Wait for home sequence completion
        IF fbMotionStage.stMotionStatus.bDone THEN
            nTestStep := 5;
        END_IF
END_CASE

fbCamSwitchPulserSearch();
fbCamSwitchPulserSync();
fbTestTimer();
fbMotionStage();

IF nTestStep = 5 THEN
    AssertTrue(
        Condition := fbAxisRef[13].Status.Homed,
        Message := 'Axis not calibrated #1'
    );
    AssertEquals_LREAL(
        Delta := 0.001,
        Expected := fbMotionStage.stMotionCommand.fHomePosition,
        Actual := fbAxisRef[13].NcToPlc.ActPos,
        Message := 'Position is not the expected #2'
    );
    TEST_FINISHED();
ELSIF fbTestTimer.Q THEN
    AssertTrue(
        Condition := FALSE,
        Message := CONCAT('Timed out at step: ', TO_STRING(nTestStep))
    );
    TEST_FINISHED();
END_IF
END_METHOD

METHOD PRIVATE GivenHomeCmdHomeViaLowModeBackwardSwPulseBeforeHomeSwPulseThenMoveToUserDefinePosition_Test15
VAR_INST
   fbMotionStage : FB_MotionStageNC(	sName := 'Test15',
                                        AxisRef := fbAxisRef[15],
                                        iPersistentDataStorage := fbPersistentDataStorage[15]
                                    ) :=(SaveAxisParams := FALSE);
									
    fbTestTimer: TON := (IN:=TRUE, PT:=T#10S);
    fbCamSwitchPulserSearch: TON := (IN:=TRUE, PT:=T#500MS);
    fbCamSwitchPulserSync: TON := (PT:=T#1000MS);
    nTestStep : INT;
END_VAR
TEST(__POUNAME());

CASE nTestStep OF
    0: // Enable all interlocks/limits for initial homing (home switch not active yet!)
        fbMotionStage.EnableLimits(
            BackwardEnable := TRUE, 
            ForwardEnable  := TRUE,
            HomeEnable     := FALSE
        );
        fbMotionStage.EnableInterlocks();
        nTestStep := 1;

    1: // Issue homing command (via high limit, should travel to positive end first)
        fbMotionStage.Home(
            HomePosition := 5.0,
            HomeMode := E_EpicsHomeCmd.HOME_VIA_LOW
        );
        nTestStep := 2;

    2: // Simulate forward limit drop
        IF fbCamSwitchPulserSearch.Q THEN
            fbMotionStage.EnableLimits(
                BackwardEnable := FALSE, 
                ForwardEnable  := TRUE,
                HomeEnable     := FALSE
            );
            fbCamSwitchPulserSearch.IN := FALSE;
            fbCamSwitchPulserSync.IN := TRUE;
            nTestStep := 3;
        END_IF

    3: // Restore forward limit after event
        IF fbCamSwitchPulserSync.Q THEN
            fbMotionStage.EnableLimits(
                BackwardEnable := TRUE, 
                ForwardEnable  := TRUE,
                HomeEnable     := FALSE
            );
            fbCamSwitchPulserSync.IN := FALSE;
            nTestStep := 4;
        END_IF

    4: // Wait for "first stage" (positive limit) homing done (i.e. LimHomeDone signals)
        IF fbMotionStage.stExMotionStatus.bLimHomeDone THEN
            // prepare for home switch pulse
            fbCamSwitchPulserSearch.IN := TRUE;
            fbCamSwitchPulserSync.IN := FALSE;
            nTestStep := 5;
        END_IF

    5: // Simulate home switch engagement (simulate HomeEnable = TRUE)
        IF fbCamSwitchPulserSearch.Q THEN
            fbMotionStage.EnableLimits(
                BackwardEnable := TRUE, 
                ForwardEnable  := TRUE,
                HomeEnable     := TRUE
            );
            fbCamSwitchPulserSearch.IN := FALSE;
            fbCamSwitchPulserSync.IN := TRUE;
            nTestStep := 6;
        END_IF

    6: // Simulate home switch disengagement (return HomeEnable to FALSE)
        IF fbCamSwitchPulserSync.Q THEN
            fbMotionStage.EnableLimits(
                BackwardEnable := TRUE, 
                ForwardEnable  := TRUE,
                HomeEnable     := FALSE
            );
            fbCamSwitchPulserSync.IN := FALSE;
            nTestStep := 7;
        END_IF 

    7: // Wait for overall homing to complete (done)
        IF fbMotionStage.stMotionStatus.bDone THEN
            nTestStep := 8;
        END_IF
END_CASE

// Cyclic calls required for timer and cam events and motion stage
fbCamSwitchPulserSearch();
fbCamSwitchPulserSync();
fbTestTimer();
fbMotionStage();

IF nTestStep = 8 THEN
    AssertTrue(
        Condition := fbAxisRef[15].Status.Homed,
        Message := 'Axis not calibrated #1'
    );
    AssertEquals_LREAL(
        Delta := 0.001,
        Expected := fbMotionStage.stMotionCommand.fHomePosition,
        Actual := fbAxisRef[15].NcToPlc.ActPos,
        Message := 'Position is not the expected #2'
    );
    TEST_FINISHED();
ELSIF fbTestTimer.Q THEN
    AssertTrue(
        Condition := FALSE,
        Message := CONCAT('Timed out at step: ', TO_STRING(nTestStep))
    );
    TEST_FINISHED();
END_IF
END_METHOD

METHOD PRIVATE GivenHomeCmdHomeViaLowModeHomeSwPulseMoveOkThenMoveToUserDefinedHomePosition_Test12
VAR_INST
   fbMotionStage : FB_MotionStageNC(	sName := 'Test12',
                                        AxisRef := fbAxisRef[12],
                                        iPersistentDataStorage := fbPersistentDataStorage[12]
                                    ) :=(SaveAxisParams := FALSE);
									
    fbTestTimer: TON := (IN:=TRUE, PT:=T#10S);
    fbCamSwitchPulserSearch: TON := (IN:=TRUE, PT:=T#500MS);
    fbCamSwitchPulserSync: TON := (PT:=T#1000MS);
    nTestStep : INT;
END_VAR
TEST(__POUNAME());

CASE nTestStep OF
    0: // Enable all interlocks/limits to be ready for homing
		fbMotionStage.EnableLimits(
			BackwardEnable:=TRUE, 
			ForwardEnable:=TRUE,
			HomeEnable:=FALSE
		);
        fbMotionStage.EnableInterlocks();
        nTestStep := 1;

    1: // Issue home command (to low limit)
        fbMotionStage.Home(HomePosition := 20.0, HomeMode := E_EpicsHomeCmd.HOME_VIA_LOW);
        nTestStep := 2;

    2: // Simulate limit switch drop/restore with cam switch events
        IF fbCamSwitchPulserSearch.Q THEN
			fbMotionStage.EnableLimits(
				BackwardEnable:=TRUE, 
				ForwardEnable:=TRUE,
				HomeEnable:=TRUE
			);
            fbCamSwitchPulserSearch.IN := FALSE;
            fbCamSwitchPulserSync.IN := TRUE;
            nTestStep := 3;
        END_IF

    3: // Restore limit after cam event
        IF fbCamSwitchPulserSync.Q THEN
			fbMotionStage.EnableLimits(
				BackwardEnable:=TRUE, 
				ForwardEnable:=TRUE,
				HomeEnable:=FALSE
			);
            nTestStep := 4;
        END_IF

    4: // Wait for home sequence completion
        IF fbMotionStage.stMotionStatus.bDone THEN
            nTestStep := 5;
        END_IF
END_CASE

fbCamSwitchPulserSearch();
fbCamSwitchPulserSync();
fbTestTimer();
fbMotionStage();

IF nTestStep = 5 THEN
    AssertTrue(
        Condition := fbAxisRef[12].Status.Homed,
        Message := 'Axis not calibrated #1'
    );
    AssertEquals_LREAL(
        Delta := 0.001,
        Expected := fbMotionStage.stMotionCommand.fHomePosition,
        Actual := fbAxisRef[12].NcToPlc.ActPos,
        Message := 'Position is not the expected #2'
    );
    TEST_FINISHED();
ELSIF fbTestTimer.Q THEN
    AssertTrue(
        Condition := FALSE,
        Message := CONCAT('Timed out at step: ', TO_STRING(nTestStep))
    );
    TEST_FINISHED();
END_IF
END_METHOD

METHOD PRIVATE GivenHomeCmdLowLimitModeAndResetThenAbortHoming_Test16
VAR_INST
   fbMotionStage : FB_MotionStageNC(	sName := 'Test16',
                                        AxisRef := fbAxisRef[16],
                                        iPersistentDataStorage := fbPersistentDataStorage[16]
                                    ):=(SaveAxisParams := FALSE);
									
    fbTestTimer: TON := (IN:=TRUE, PT:=T#3S);
    fbResetTimer: TON := (IN:=TRUE, PT:=T#500MS);
    nTestStep : INT;
END_VAR
TEST(__POUNAME());


CASE nTestStep OF
    0: // Enable all interlocks/limits for initial homing (home switch not active yet!)
        fbMotionStage.EnableLimits(
            BackwardEnable := TRUE, 
            ForwardEnable  := TRUE,
            HomeEnable     := FALSE
        );
        fbMotionStage.EnableInterlocks();
        nTestStep := 1;

    1: // Issue homing command (via high limit, should travel to positive end first)
        fbMotionStage.Home(
            HomePosition := 5.0,
            HomeMode := E_EpicsHomeCmd.LOW_LIMIT
        );
        nTestStep := 2;
    2:
        IF fbResetTimer.Q THEN
            fbMotionStage.Reset();
            fbResetTimer.IN := FALSE;
            nTestStep := 3;
        END_IF
    3:
		// resetting a homing sequence will set mc_home into error state
        IF fbMotionStage.stMotionStatus.bDone THEN
            nTestStep := 4;
        END_IF
END_CASE

fbResetTimer();
fbTestTimer();
fbMotionStage();

IF nTestStep = 4 THEN
    TEST_FINISHED();
ELSIF fbTestTimer.Q THEN
    AssertTrue(
        Condition := FALSE,
        Message := CONCAT('Timed out at step: ', TO_STRING(nTestStep))
    );

    TEST_FINISHED();
END_IF
END_METHOD

METHOD PRIVATE GivenHomeCmdLowLimitModeBackwardSwPulseMoveOkThenMoveToUserDefinedHomePosition_Test10
VAR_INST
   fbMotionStage : FB_MotionStageNC(	sName := 'Test10',
                                        AxisRef := fbAxisRef[10],
                                        iPersistentDataStorage := fbPersistentDataStorage[10]
                                    ):=(SaveAxisParams := FALSE);
									
    fbTestTimer: TON := (IN:=TRUE, PT:=T#10S);
    fbCamSwitchPulserSearch: TON := (IN:=TRUE, PT:=T#500MS);
    fbCamSwitchPulserSync: TON := (PT:=T#1000MS);
    nTestStep : INT;
END_VAR
TEST(__POUNAME());

CASE nTestStep OF
    0: // Enable all interlocks/limits to be ready for homing
        fbMotionStage.EnableLimits(
			BackwardEnable:=TRUE, 
			ForwardEnable:=TRUE,
			HomeEnable:=FALSE
		);
        fbMotionStage.EnableInterlocks();
        nTestStep := 1;

    1: // Issue home command (to low limit)
        fbMotionStage.Home(HomePosition := 20.0, HomeMode := E_EpicsHomeCmd.LOW_LIMIT);
        nTestStep := 2;

    2: // Simulate limit switch drop/restore with cam switch events
		// simulate limit release
        IF fbCamSwitchPulserSearch.Q THEN
			fbMotionStage.EnableLimits(
				BackwardEnable:=FALSE, 
				ForwardEnable:=TRUE,
				HomeEnable:=FALSE
			);
            fbCamSwitchPulserSearch.IN := FALSE;
            fbCamSwitchPulserSync.IN := TRUE;
            nTestStep := 3;
        END_IF

    3: // Restore limit after cam event
        IF fbCamSwitchPulserSync.Q THEN
			fbMotionStage.EnableLimits(
				BackwardEnable:=TRUE, 
				ForwardEnable:=TRUE,
				HomeEnable:=FALSE
			);
            nTestStep := 4;
        END_IF

    4: // Wait for home sequence completion
        IF fbMotionStage.stMotionStatus.bDone THEN
            nTestStep := 5;
        END_IF
END_CASE

fbCamSwitchPulserSearch();
fbCamSwitchPulserSync();
fbTestTimer();
fbMotionStage();

IF nTestStep = 5 THEN
    AssertTrue(
        Condition := fbAxisRef[10].Status.Homed,
        Message := 'Axis not calibrated #1'
    );
    AssertEquals_LREAL(
        Delta := 0.001,
        Expected := fbMotionStage.stMotionCommand.fHomePosition,
        Actual := fbAxisRef[10].NcToPlc.ActPos,
        Message := 'Position is not the expected #2'
    );
    TEST_FINISHED();
ELSIF fbTestTimer.Q THEN
    AssertTrue(
        Condition := FALSE,
        Message := CONCAT('Timed out at step: ', TO_STRING(nTestStep))
    );
    TEST_FINISHED();
END_IF
END_METHOD

METHOD PRIVATE GivenHomeCmdNoneAndMoveOkThenSetHomeFlag_Test9
VAR_INST
   fbMotionStage : FB_MotionStageNC(	sName := 'Test9',
                                        AxisRef := fbAxisRef[9],
                                        iPersistentDataStorage := fbPersistentDataStorage[9]
                                    ):=(SaveAxisParams := FALSE);
									
    fbTestTimer: TON := (IN:=TRUE, PT:=T#3S);
    nTestStep : INT;
END_VAR
TEST(__POUNAME());


CASE nTestStep OF
    0:
		// Enable safety interlocks and hardware limits
        fbMotionStage.EnableLimits(
			BackwardEnable:=TRUE, 
			ForwardEnable:=TRUE,
			HomeEnable:=FALSE
		);
        fbMotionStage.EnableInterlocks();
		nTestStep := 1;
	1:
		fbMotionStage.Home(HomePosition:=20.0, HomeMode:=E_EPicsHomeCmd.NONE);
		nTestStep := 2;
	2:
		IF fbMotionStage.stMotionStatus.bHomed THEN
			nTestStep := 3;
		END_IF	
END_CASE

fbTestTimer();
fbMotionStage();

IF nTestStep = 3 THEN

TEST_FINISHED();
ELSIF fbTestTimer.Q THEN
    AssertTrue(
        Condition := FALSE,
        Message := CONCAT('Timed out at step: ', TO_STRING(nTestStep))
    );
    TEST_FINISHED();
END_IF
END_METHOD

METHOD PRIVATE GivenMoveCmdAndMoveOkAndNegativeBacklashEnabledThenMoveToTargetWithCompensation_Test7
VAR_INST
   fbMotionStage : FB_MotionStageNC(	sName := 'Test7',
                                        AxisRef := fbAxisRef[7],
                                        iPersistentDataStorage := fbPersistentDataStorage[7]
                                    ):=(SaveAxisParams := FALSE);
									
    fbTestTimer: TON := (IN:=TRUE, PT:=T#10S);
    nTestStep : INT;
END_VAR
TEST(__POUNAME());

CASE nTestStep OF
    0: // Enable safety and backlash compensation
         fbMotionStage.EnableLimits(
			BackwardEnable:=TRUE, 
			ForwardEnable:=TRUE,
			HomeEnable:=FALSE
		);
        fbMotionStage.EnableInterlocks();
		fbMotionStage.EnableBacklashCompensation(UserEnable := TRUE, Compensation := -2.5);
        nTestStep := 1;
    1: // Forward move, should have **no** compensation applied
        fbMotionStage.AbsoluteMoveWithBacklashCompensation(
            Position := -10.0,
            Velocity := 200.0,
            Acceleration := 400.0,
            Deceleration := 400.0
        );
        nTestStep := 2;
    2:
        IF fbMotionStage.stMotionStatus.bDone THEN
            AssertTrue(
                Condition := ABS(-10.0 - fbAxisRef[7].NcToPlc.ActPos) < 0.001,
                Message := 'Target position not reached #1'
            );
            AssertTrue(
                Condition := (fbAxisRef[7].NcToPlc.ActPos - fbAxisRef[7].NcToPlc.ActPosWithoutPosCorrection) = 0,
                Message := 'No compensation in this direction #2'
            );
            nTestStep := 3;
        END_IF
    3: // Reverse move, should have 2.5 compensation
        fbMotionStage.AbsoluteMoveWithBacklashCompensation(
            Position := 80.0,
            Velocity := 200.0,
            Acceleration := 400.0,
            Deceleration := 400.0
        );
        nTestStep := 4;
    4:
        IF fbMotionStage.stMotionStatus.bDone THEN
            AssertTrue(
                Condition := ABS(80.0 - fbAxisRef[7].NcToPlc.ActPos) < 0.001,
                Message := 'Target position not reached #3'
            );
            AssertTrue(
                Condition := (fbAxisRef[7].NcToPlc.ActPos - fbAxisRef[7].NcToPlc.ActPosWithoutPosCorrection) = 2.5,
                Message := 'This move must have a 2.5 compensation #4'
            );
            nTestStep := 5;
        END_IF
    5: // Compensation now 0, move uncompensated
        fbMotionStage.EnableBacklashCompensation(UserEnable := TRUE, Compensation := 0);
        nTestStep := 6;
    6:
        fbMotionStage.AbsoluteMoveWithBacklashCompensation(
            Position := 120.0,
            Velocity := 200.0,
            Acceleration := 400.0,
            Deceleration := 400.0
        );
        nTestStep := 7;
    7:
        IF fbMotionStage.stMotionStatus.bDone THEN
            AssertTrue(
                Condition := ABS(120.0 - fbAxisRef[7].NcToPlc.ActPos) < 0.001,
                Message := 'Target position not reached #5'
            );
            AssertTrue(
                Condition := (fbAxisRef[7].NcToPlc.ActPos - fbAxisRef[7].NcToPlc.ActPosWithoutPosCorrection) = 0,
                Message := 'Actual compensation must be 0 #6'
            );
            nTestStep := 8;
        END_IF
    8: // Set -3.5 for next, expect 3.5 compensation in reverse
        fbMotionStage.EnableBacklashCompensation(UserEnable := TRUE, Compensation := -3.5);
        nTestStep := 9;
    9:
        fbMotionStage.AbsoluteMove(
            Position := 160.0,
            Velocity := 200.0,
            Acceleration := 400.0,
            Deceleration := 400.0
        );
        nTestStep := 10;
    10:
        IF fbMotionStage.stMotionStatus.bDone THEN
            AssertTrue(
                Condition := ABS(160.0 - fbAxisRef[7].NcToPlc.ActPos) < 0.001,
                Message := 'Target position not reached #7'
            );
            AssertTrue(
                Condition := (fbAxisRef[7].NcToPlc.ActPos - fbAxisRef[7].NcToPlc.ActPosWithoutPosCorrection) = 3.5,
                Message := 'This move must have a 3.5 compensation #8'
            );
            nTestStep := 11;
        END_IF
    11: // Disable compensation, next should be uncompensated
        fbMotionStage.EnableBacklashCompensation(UserEnable := FALSE, Compensation := -3.5);
        nTestStep := 12;
    12:
        fbMotionStage.AbsoluteMove(
            Position := 180.0,
            Velocity := 200.0,
            Acceleration := 400.0,
            Deceleration := 400.0
        );
        nTestStep := 13;
    13:
        IF fbMotionStage.stMotionStatus.bDone THEN
            AssertTrue(
                Condition := ABS(180.0 - fbAxisRef[7].NcToPlc.ActPos) < 0.001,
                Message := 'Target position not reached #9'
            );
            AssertTrue(
                Condition := (fbAxisRef[7].NcToPlc.ActPos - fbAxisRef[7].NcToPlc.ActPosWithoutPosCorrection) = 0,
                Message := 'This move is not compensated #10'
            );
            nTestStep := 14;
        END_IF
END_CASE

fbTestTimer();
fbMotionStage();

IF nTestStep = 14 THEN
    TEST_FINISHED();
ELSIF fbTestTimer.Q THEN
    AssertTrue(
        Condition := FALSE,
        Message := CONCAT('Timed out at step: ', TO_STRING(nTestStep))
    );
    TEST_FINISHED();
END_IF
END_METHOD

METHOD PRIVATE GivenMoveCmdAndMoveOkAndPositiveBacklashEnabledThenMoveToTargetWithCompensation_Test6
VAR_INST
   fbMotionStage : FB_MotionStageNC(	sName := 'Test6',
                                        AxisRef := fbAxisRef[6],
                                        iPersistentDataStorage := fbPersistentDataStorage[6]
                                    ) :=(SaveAxisParams := FALSE);
									
    fbTestTimer: TON := (IN:=TRUE, PT:=T#10S);
    nTestStep : INT;
END_VAR
TEST(__POUNAME());

CASE nTestStep OF
    0: 
		//Enable safety interlocks AND hardware limits
         fbMotionStage.EnableLimits(
			BackwardEnable:=TRUE, 
			ForwardEnable:=TRUE,
			HomeEnable:=FALSE
		);
		// disable restore saved position
        fbMotionStage.EnableInterlocks();
		//Enable 2.5 backlash compensation
        fbMotionStage.EnableBacklashCompensation(UserEnable := TRUE, Compensation := 2.5);
        nTestStep := 1;
    1: // Forward move, should have **no** compensation applied
        fbMotionStage.AbsoluteMoveWithBacklashCompensation(
            Position := 100.0,
            Velocity := 50.0,
            Acceleration := 500.0,
            Deceleration := 500.0
        );
        nTestStep := 2;
    2: // Wait for move done, check result
        IF fbMotionStage.stMotionStatus.bDone THEN
            AssertTrue(
                Condition := ABS(fbMotionStage.MotionCmd.fPosition - fbAxisRef[6].NcToPlc.ActPos) < 0.001,
                Message := 'Target position not reached #1'
            );
            AssertTrue(
                Condition := (fbAxisRef[6].NcToPlc.ActPos - fbAxisRef[6].NcToPlc.ActPosWithoutPosCorrection) = 0,
                Message := 'No compensation in this direction #2'
            );
            nTestStep := 3;
        END_IF
    3: // Reverse move, should have 2.5 compensation applied
        IF fbMotionStage.ExMotionStatus.bIdling THEN
            fbMotionStage.AbsoluteMoveWithBacklashCompensation(
                Position := 50.0,
                Velocity := 50.0,
                Acceleration := 500.0,
                Deceleration := 500.0
            );
            nTestStep := 4;
        END_IF
    4:
        IF fbMotionStage.stMotionStatus.bDone THEN
            AssertTrue(
                Condition := ABS(fbMotionStage.MotionCmd.fPosition - fbAxisRef[6].NcToPlc.ActPos) < 0.001,
                Message := 'Target position not reached #3'
            );
            AssertTrue(
                Condition := ((fbAxisRef[6].NcToPlc.ActPos - fbAxisRef[6].NcToPlc.ActPosWithoutPosCorrection)- 2.5) < 0.001,
                Message := 'This move must have a 2.5 compensation #4'
            );
            nTestStep := 5;
        END_IF
    5: // Set compensation to 0, next move should be uncompensated
        fbMotionStage.EnableBacklashCompensation(UserEnable := TRUE, Compensation := 0);
        nTestStep := 6;
    6:
        fbMotionStage.AbsoluteMoveWithBacklashCompensation(
            Position := 60.0,
            Velocity := 50.0,
            Acceleration := 200.0,
            Deceleration := 200.0
        );
        nTestStep := 7;
    7:
        IF fbMotionStage.stMotionStatus.bDone THEN
            AssertTrue(
                Condition := ABS(60.0 - fbAxisRef[6].NcToPlc.ActPos) < 0.001,
                Message := 'Target position not reached #5'
            );
            AssertTrue(
                Condition := (fbAxisRef[6].NcToPlc.ActPos - fbAxisRef[6].NcToPlc.ActPosWithoutPosCorrection) = 0,
                Message := 'Actual compensation must be 0 #6'
            );
            nTestStep := 8;
        END_IF
    8: // Set comp to 3.5 for next move
        fbMotionStage.EnableBacklashCompensation(UserEnable := TRUE, Compensation := 3.5);
        nTestStep := 9;
    9:
        fbMotionStage.AbsoluteMoveWithBacklashCompensation(
            Position := 40.0,
            Velocity := 50.0,
            Acceleration := 200.0,
            Deceleration := 200.0
        );
        nTestStep := 10;
    10:
        IF fbMotionStage.stMotionStatus.bDone THEN
            AssertTrue(
                Condition := ABS(40.0 - fbAxisRef[6].NcToPlc.ActPos) < 0.001,
                Message := 'Target position not reached #7'
            );
            AssertTrue(
                Condition := ((fbAxisRef[6].NcToPlc.ActPos - fbAxisRef[6].NcToPlc.ActPosWithoutPosCorrection)- 3.5) < 0.001,
                Message := 'This move must have a 3.5 compensation #8'
            );
            nTestStep := 11;
        END_IF
    11: // Disable compensation, next move should show 0 compensation
        fbMotionStage.EnableBacklashCompensation(UserEnable := FALSE, Compensation := 0.5);
        nTestStep := 12;
    12:
        fbMotionStage.AbsoluteMoveWithBacklashCompensation(
            Position := 20.0,
            Velocity := 50.0,
            Acceleration := 200.0,
            Deceleration := 200.0
        );
        nTestStep := 13;
    13:
        IF fbMotionStage.stMotionStatus.bDone THEN
            AssertTrue(
                Condition := ABS(20.0 - fbAxisRef[6].NcToPlc.ActPos) < 0.001,
                Message := 'Target position not reached #9'
            );
            AssertTrue(
                Condition := (fbAxisRef[6].NcToPlc.ActPos - fbAxisRef[6].NcToPlc.ActPosWithoutPosCorrection) = 0,
                Message := 'This move is not compensated #10'
            );
            nTestStep := 14;
        END_IF
END_CASE

fbTestTimer();
fbMotionStage();

IF nTestStep = 14 THEN
    TEST_FINISHED();
ELSIF fbTestTimer.Q THEN
    AssertTrue(
        Condition := FALSE,
        Message := CONCAT('Timed out at step: ', TO_STRING(nTestStep))
    );
    TEST_FINISHED();
END_IF
END_METHOD

METHOD PRIVATE GivenMoveCmdAndMoveOkIfHaltThenAbortMove_Test2
VAR_INST
   fbMotionStage : FB_MotionStageNC(	sName := 'Test2',
                                        AxisRef := fbAxisRef[2],
                                        iPersistentDataStorage := fbPersistentDataStorage[2]
                                    ) :=(SaveAxisParams := FALSE);
									
    fbTestTimer: TON := (IN:=TRUE, PT:=T#3S);
    fbAbsoluteMoveHaltTimer: TON := (PT:=T#100MS);
    nTestStep : INT;
END_VAR
TEST(__POUNAME());

fbMotionStage(); // Call stage logic cyclically

// State machine for staged assertions
CASE nTestStep OF
    // Interlock error check
    0:
        IF fbMotionStage.ExMotionStatus.bInterlocksError THEN
            AssertTrue(
                Condition := fbMotionStage.stMotionStatus.bError,
                Message   := 'Interlock error must be raised #2'
            );
            AssertEquals_UDINT(
                Expected := 11,
                Actual   := fbMotionStage.stMotionStatus.nErrorId,
                Message  := 'Interlock error code is 11 #3'
            );		
        END_IF
        nTestStep := 1;

    // Reset, enable limits and interlocks
    1:
        fbMotionStage.Reset();
        fbMotionStage.EnableLimits(
			BackwardEnable:=TRUE, 
			ForwardEnable:=TRUE,
			HomeEnable:=FALSE
		);
        fbMotionStage.EnableInterlocks();
        // Compiler shouldn't allow property set if property is get-only 
        // (review behavior: see your original comments).
        nTestStep := 2;	

    // After abort, error should be cleared
    2:
        IF fbMotionStage.ExMotionStatus.bAbortDone THEN
            AssertFalse(
                Condition := fbMotionStage.stMotionStatus.bError,
                Message   := 'Error must cleared #4'
            );
            AssertEquals_UDINT(
                Expected := 0,
                Actual   := fbMotionStage.stMotionStatus.nErrorId,
                Message  := 'error ID must 0 #5'
            );
            nTestStep := 3;	
        END_IF

    // Command an absolute move
    3:
        fbMotionStage.AbsoluteMove(
            Position := 1000.0,
            Velocity := 50.0,
            Acceleration := 200.0,
            Deceleration := 200.0
        );
        fbAbsoluteMoveHaltTimer.IN := TRUE;
        nTestStep := 4;

    // After short timer, send Halt
    4:
        IF fbAbsoluteMoveHaltTimer.Q THEN
            fbMotionStage.Halt();
            fbAbsoluteMoveHaltTimer.IN := FALSE;
            nTestStep := 5;
        END_IF

